Yaskawa INFORM job: OK_R2_O38-47,64(2)(90,0)_HARDOX.JBI

/JOB
//NAME OK_R2_O38-47,64(2)(90,0)_HARDOX
///FOLDERNAME X4
//POS
///NPOS 526,526,526,27,0,0
///TOOL 0
///POSTYPE PULSE
///PULSE
C00000=-102904,-190754,-108658,-56793,33718,43054
C00001=-112112,-124440,-79629,-37912,40591,30924
C00002=-145621,-43895,-45824,-14341,74181,8322
C00003=-153971,-33006,-36006,-12070,72386,5523
C00004=-155060,-28858,-31777,-11788,71762,5195
C00005=-155060,-28697,-30772,-11821,71236,5249
C00006=-155060,-28799,-31389,-11800,71558,5216
C00007=-155039,-34474,-35187,-11843,70998,5279
C00008=-155039,-34310,-34280,-11875,70534,5325
C00009=-155401,-30968,-32059,-11745,70828,5164
C00010=-155377,-31193,-32210,-11754,70809,5175
C00011=-155377,-31138,-31906,-11765,70652,5191
C00012=-155377,-31202,-32269,-11753,70839,5173
C00013=-155039,-34366,-34582,-11864,70687,5310
C00014=-155039,-34238,-33894,-11889,70337,5345
C00015=-155199,-32420,-32682,-11831,70497,5273
C00016=-155039,-34561,-35687,-11827,71256,5253
C00017=-155039,-34852,-37545,-11764,60729,-61899
C00018=-154233,-9766,-49045,-10778,79336,-63369
C00019=-160860,20388,-27147,4890,89580,-62573
C00020=-159005,21387,-26719,10091,95401,40718
C00021=-157683,11153,-31727,14818,95267,42221
C00022=-157333,10978,-31290,14718,94862,42282
C00023=-157333,10579,-30718,14700,94322,42218
C00024=-157333,10654,-30827,14702,94424,42231
C00025=-157208,13112,-28644,14670,94325,42258
C00026=-157333,10654,-30827,14702,94424,42231
C00027=-155197,18382,-25631,10360,99317,42541
C00028=-156128,18351,-25710,10541,99457,42258
C00029=-155197,18405,-25661,10361,99347,42543
C00030=-157150,29334,-18312,13637,104284,-74335
C00031=-160757,60877,11500,15991,103565,-75216
C00032=-161248,60365,12974,15966,102528,-75520
C00033=-161248,59958,13544,15927,101988,-75592
C00034=-161248,60034,13428,15935,102095,-75578
C00035=-161237,57406,10441,15969,102563,-75510
C00036=-161248,60034,13428,15935,102095,-75578
C00037=-165275,44513,292,24456,94477,-76762
C00038=-164215,44651,439,24212,94172,-76462
C00039=-165275,45390,-990,24520,95610,-76527
C00040=-163079,30136,-11541,1568,89602,-59565
C00041=-168249,10711,-29896,3021,91050,-61145
C00042=-157831,-12146,-38438,-15492,88791,-34391
C00043=-155039,-34561,-35687,-11827,71256,5253
C00044=-150032,-44426,-43245,-13273,71622,7027
C00045=-145621,-43895,-45824,-14341,74181,8322
C00046=-126188,-124725,-79701,-29915,35046,24780
C00047=-126055,-123557,-80227,-30584,36919,-46840
C00048=-134159,-82950,-60455,-26786,53755,-58167
C00049=-139895,-66772,-53027,-23260,55430,-61177
C00050=-141080,-64871,-50726,-22849,54691,-61528
C00051=-141080,-64256,-48906,-23069,53949,-61354
C00052=-141080,-64445,-49458,-23002,54172,-61405
C00053=-141699,-58855,-46559,-22430,55006,-61872
C00054=-141699,-58644,-45888,-22510,54724,-61808
C00055=-141384,-60956,-47106,-22771,54406,-61595
C00056=-141666,-61047,-48744,-22388,55219,-61905
C00057=-175822,-56342,-55375,-14128,52086,-76708
C00058=-175822,-56190,-54452,-14221,51611,-76640
C00059=-175822,-55829,-52499,-14419,50624,-76498
C00060=-175822,-55911,-52925,-14375,50838,-76529
C00061=-175468,-48992,-48997,-14371,52005,-76544
C00062=-175468,-48914,-48510,-14420,51752,-76509
C00063=-175508,-50972,-49701,-14458,51431,-76479
C00064=-175513,-50711,-51459,-14225,52610,-76651
C00065=-145967,-74518,-63848,-31232,56636,-64447
C00066=-145831,-74953,-63116,-31520,56106,-64204
C00067=-145831,-74483,-61568,-31767,55497,-64004
C00068=-145831,-74555,-61804,-31730,55589,-64033
C00069=-146027,-71690,-60453,-31425,56067,-64284
C00070=-145831,-74555,-61804,-31730,55589,-64033
C00071=-144274,-73926,-61511,-32332,56303,-63536
C00072=-142723,-73317,-61225,-32917,57019,-63047
C00073=-144274,-74241,-62562,-32164,56716,-63675
C00074=-154468,-41208,-54710,-20041,83622,-74370
C00075=-154754,-41232,-53805,-19994,83017,-74368
C00076=-154754,-41278,-52810,-20016,82420,-74271
C00077=-154754,-41268,-53081,-20010,82580,-74296
C00078=-154720,-44115,-54834,-20034,82227,-74224
C00079=-154754,-41268,-53081,-20010,82580,-74296
C00080=-155675,-41399,-53162,-19802,82346,-74583
C00081=-157197,-41522,-53239,-19453,81973,-75060
C00082=-155675,-41327,-54458,-19774,83133,-74712
C00083=-153395,-74759,-74503,-20498,79124,-73228
C00084=-153314,-74128,-71798,-20600,77886,-72984
C00085=-153314,-73934,-70558,-20645,77263,-72875
C00086=-153314,-73981,-70840,-20635,77403,-72900
C00087=-153337,-77229,-72353,-20684,76704,-72788
C00088=-153314,-73981,-70840,-20635,77403,-72900
C00089=-154242,-74168,-70928,-20438,77132,-73193
C00090=-156115,-74593,-71128,-20032,76581,-73782
C00091=-154242,-74289,-71704,-20409,77523,-73260
C00092=-153903,-106822,-81190,-17417,50996,-69253
C00093=-154273,-105923,-79990,-17297,50655,-69359
C00094=-154273,-105262,-78653,-17414,50193,-69275
C00095=-154273,-105373,-78877,-17395,50270,-69289
C00096=-154522,-102445,-77859,-17058,51058,-69542
C00097=-154273,-105373,-78877,-17395,50270,-69289
C00098=-152960,-105275,-78843,-18047,50584,-68754
C00099=-150354,-104788,-78676,-19283,51319,-67719
C00100=-152960,-106026,-80369,-17910,51111,-68853
C00101=-102904,-190754,-108658,-56793,33718,43054
C00102=-131529,-189509,-110128,-36771,24434,27261
C00103=-124211,-86804,-80218,-19393,77786,15538
C00104=-160160,17664,-548,-10057,75687,3034
C00105=-160660,22954,7322,-10002,73531,3037
C00106=-166196,35697,21074,-8411,71011,1264
C00107=-166196,35823,21925,-8432,70556,1296
C00108=-166196,35779,21629,-8424,70714,1284
C00109=-166257,29532,15350,-8374,71357,1216
C00110=-166257,29595,15824,-8387,71101,1234
C00111=-166146,32147,18367,-8436,70861,1292
C00112=-166154,31970,18190,-8433,70878,1288
C00113=-166154,32007,18455,-8439,70734,1299
C00114=-166154,31970,18190,-8433,70878,1288
C00115=-166179,28892,15129,-8411,71174,1259
C00116=-166179,28962,15640,-8424,70899,1278
C00117=-166104,30948,17607,-8456,70718,1318
C00118=-166176,28573,11657,-8324,73127,1123
C00119=-182178,81885,43168,-17852,83199,-7398
C00120=-187829,78862,41539,-16297,81531,-9102
C00121=-187829,78684,42370,-16320,80951,-9022
C00122=-187829,78533,43217,-16344,80374,-8946
C00123=-187829,78564,43028,-16338,80502,-8962
C00124=-188354,71817,34916,-16132,81866,-9324
C00125=-188354,71755,35176,-16139,81682,-9298
C00126=-188062,74943,38982,-16246,81057,-9118
C00127=-188087,74664,38647,-16237,81113,-9134
C00128=-188087,74606,38940,-16246,80911,-9107
C00129=-188087,74636,38787,-16240,81016,-9121
C00130=-188430,70936,34375,-16113,81733,-9334
C00131=-188430,70865,34684,-16121,81516,-9305
C00132=-188196,73082,37320,-16205,81097,-9170
C00133=-188430,71276,33065,-16084,82678,-9458
C00134=-165319,19573,3695,-8574,73487,1399
C00135=-163582,7043,-11027,-8999,76267,1804
C00136=-162101,-9402,-41897,-5301,86162,910
C00137=-133469,39121,-1061,931,85072,6891
C00138=-135751,46408,8355,1655,83056,6142
C00139=-135516,49476,14058,1587,81119,6193
C00140=-135516,49311,14679,1588,80652,6188
C00141=-135036,46950,11602,1434,81323,6352
C00142=-134946,46723,11962,1405,80982,6377
C00143=-135074,47950,13285,1445,80801,6333
C00144=-135102,44394,8734,1452,81774,6335
C00145=-133469,39121,-1061,931,85072,6891
C00146=-135146,16919,-22910,1456,87131,6386
C00147=-160578,-137207,-111137,27103,45167,-7155
C00148=-166532,-153428,-115250,33739,42272,-11545
C00149=-166532,-153428,-115250,33739,42272,-11545
C00150=-160883,-131526,-133102,-3483,78120,-6366
C00151=-103370,-159686,-136025,-1765,64172,-8056
C00152=-97179,-138237,-129333,-10238,76593,11306
C00153=-96065,-128281,-122439,-10507,77596,11607
C00154=-96065,-128106,-120653,-10546,76604,11690
C00155=-96065,-128281,-122439,-10507,77596,11607
C00156=-96974,-121186,-120234,-10189,79734,11117
C00157=-96065,-128281,-122439,-10507,77596,11607
C00158=-80019,-98046,-111669,-14399,88698,15911
C00159=-80077,-97852,-111516,-14385,88694,15892
C00160=-80077,-98331,-110658,-14385,87944,15982
C00161=-80077,-97897,-111441,-14385,88627,15900
C00162=-80867,-94680,-110202,-14197,89359,15553
C00163=-80077,-97897,-111441,-14385,88627,15900
C00164=-77060,-103837,-123440,-15157,93336,16325
C00165=-77104,-103620,-123385,-15148,93404,16303
C00166=-82212,-117279,-126602,-8714,87753,18646
C00167=-83304,-119533,-127995,-7425,87342,19011
C00168=-83304,-120285,-126924,-7427,86307,19072
C00169=-83304,-120125,-127175,-7427,86540,19060
C00170=-84285,-114583,-125380,-7184,88184,18645
C00171=-83304,-120125,-127175,-7427,86540,19060
C00172=-78124,-131037,-133000,-8681,85036,20864
C00173=-78124,-131037,-133000,-8681,85036,20864
C00174=-80781,-132367,-131851,-8063,83392,20088
C00175=-80781,-132658,-130737,-8071,82565,20142
C00176=-80781,-132579,-131090,-8068,82820,20125
C00177=-82215,-124520,-128659,-7695,85306,19491
C00178=-80136,-136061,-133167,-8229,82377,20371
C00179=-80218,-134686,-135534,-8183,84509,20204
C00180=-75563,-118157,-129697,-13391,92336,27261
C00181=-84024,-123631,-127734,-11595,87159,24981
C00182=-84024,-123979,-126960,-11598,86516,25042
C00183=-84024,-123746,-127494,-11596,86956,25000
C00184=-85048,-122093,-126977,-11373,87337,24623
C00185=-81994,-135324,-132084,-12059,84184,25946
C00186=-81994,-133752,-136174,-12028,87438,25630
C00187=-81994,-133752,-136174,-12028,87438,25630
C00188=-83107,-120864,-125937,-11789,87596,25245
C00189=-83880,-119254,-122492,-11630,86222,25116
C00190=-83880,-119583,-121326,-11637,85351,25197
C00191=-83880,-119399,-122020,-11633,85865,25149
C00192=-85062,-113328,-120022,-11369,87556,24598
C00193=-83880,-119399,-122020,-11633,85865,25149
C00194=-83464,-119333,-123502,-11716,86850,25194
C00195=-84085,-116294,-122008,-11580,87393,24935
C00196=-84085,-116863,-120480,-11583,86184,25047
C00197=-84085,-116689,-121008,-11580,86590,25010
C00198=-85140,-111307,-119205,-11348,88071,24523
C00199=-84085,-116194,-122230,-11576,87577,24918
C00200=-82864,-118268,-130611,-11862,91757,24924
C00201=-82864,-118268,-130611,-11862,91757,24924
C00202=-86851,-110557,-120071,-10968,88745,23893
C00203=-86851,-111341,-118540,-10968,87421,24011
C00204=-86851,-110811,-119621,-10968,88345,23929
C00205=-88598,-109546,-119189,-10575,88500,23337
C00206=-86851,-110811,-119621,-10968,88345,23929
C00207=-83825,-124590,-131318,-11630,88867,24881
C00208=-82909,-127853,-136097,-11834,90233,25054
C00209=-84148,-125178,-125504,-11579,85018,25131
C00210=-81186,-118241,-121828,-12198,86718,25964
C00211=-81186,-118533,-120824,-12201,85966,26037
C00212=-81186,-118483,-121017,-12200,86107,26023
C00213=-82314,-113243,-119285,-11952,87535,25506
C00214=-81186,-118241,-121828,-12198,86718,25964
C00215=-87931,-140644,-131144,-10841,80108,24284
C00216=-89960,-139833,-128047,-10433,78377,23732
C00217=-89960,-139550,-127065,-10448,77925,23770
C00218=-89960,-139622,-127307,-10444,78035,23761
C00219=-90753,-134395,-125809,-10209,79670,23349
C00220=-89456,-143397,-129529,-10578,77538,23979
C00221=-95203,-107502,-133483,-6717,98684,21003
C00222=-95203,-107502,-133483,-6717,98684,21003
C00223=70091,-137861,-134613,19540,89589,-11549
C00224=70091,-137861,-134613,19540,89589,-11549
C00225=89914,-142582,-130695,14485,81723,-10120
C00226=90202,-137048,-128128,14398,82897,-9883
C00227=90202,-136718,-126391,14423,82025,-9985
C00228=90202,-136862,-127082,14413,82365,-9945
C00229=91010,-131454,-125503,14223,83978,-9478
C00230=90202,-137070,-128271,14397,82970,-9874
C00231=76195,-137070,-128271,14397,82970,-9874
C00232=74994,-123934,-123423,14560,86840,-9835
C00233=74994,-124092,-122198,14564,86029,-9931
C00234=74994,-124005,-122955,14561,86525,-9872
C00235=76141,-119465,-121513,14342,87728,-9340
C00236=72631,-133219,-128550,14998,85696,-10781
C00237=72631,-131663,-134232,14989,89852,-10278
C00238=50716,-132590,-134806,14983,95067,-21778
C00239=53786,-122460,-125023,14607,93736,-20890
C00240=54881,-121663,-124068,14472,93371,-20558
C00241=54881,-122014,-122728,14450,92397,-20672
C00242=54881,-121856,-123398,14460,92875,-20616
C00243=56721,-117465,-121986,14267,93906,-19868
C00244=54881,-121856,-123398,14460,92875,-20616
C00245=55322,-120745,-123309,14420,93300,-20415
C00246=55322,-120747,-123302,14420,93295,-20416
C00247=55322,-120978,-122461,14407,92679,-20487
C00248=55322,-120864,-122902,14414,92999,-20450
C00249=56710,-117554,-121835,14266,93775,-19889
C00250=54436,-122887,-123768,14509,92662,-20793
C00251=54436,-122067,-126198,14556,94519,-20574
C00252=53688,-126302,-127242,14482,93230,-21000
C00253=7968,-117738,-135568,14910,102458,-19890
C00254=7968,-117738,-135568,14910,102458,-19890
C00255=4119,-116606,-125698,15061,97809,-21757
C00256=7770,-114903,-122318,14590,96007,-20739
C00257=7770,-115418,-121244,14557,95111,-20843
C00258=7770,-115024,-122084,14598,95810,-20761
C00259=9375,-110655,-120613,14452,96836,-20097
C00260=7770,-115024,-122084,14598,95810,-20761
C00261=10569,-102485,-118509,17167,107955,-30726
C00262=17008,-101176,-116544,17116,107524,-30934
C00263=-121481,-92648,-105286,-5369,115019,-86755
C00264=-120615,-96829,-107734,-5213,114434,-86412
C00265=23859,-150611,-131722,11614,81196,-13147
C00266=5605,-98558,-114313,9016,91646,-19053
C00267=5292,-97369,-113802,9089,91971,-19129
C00268=5881,-109040,-123705,8960,92007,-18939
C00269=6434,-120006,-133010,8839,92040,-18760
C00270=-12667,-120051,-129788,-19636,91452,63850
C00271=-15640,-171133,-136982,-20070,70138,66271
C00272=3779,-163113,-125940,-36463,74354,73480
C00273=-120436,-95190,-80290,-14692,43277,16053
C00274=-119715,-95468,-78930,-15521,42464,16563
C00275=1349,-140937,-118482,-38247,78517,71026
C00276=-15636,-141614,-117585,-35447,65083,67762
C00277=-17609,-126505,-112505,-34601,67163,66072
C00278=-24043,-118481,-124771,-21586,79008,61529
C00279=-24043,-118481,-124771,-21586,79008,61529
C00280=-75030,-118005,-124618,-21594,79160,61521
C00281=-115715,-153549,-128562,15788,54400,49074
C00282=-122131,-153692,-122292,24372,49463,44977
C00283=-120438,-96789,-101713,-1489,48968,3516
C00284=-120356,-99154,-104149,-1548,49253,3547
C00285=-84198,-116806,-111213,1772,54897,61304
C00286=-87160,-120534,-109364,10018,48087,58269
C00287=-90828,-138253,-118809,13315,45388,56216
C00288=-90828,-138253,-118809,13315,45388,56216
C00289=-90828,-142934,-129815,12421,49655,56806
C00290=-90829,-142933,-129813,12421,49658,56806
C00291=-119872,-163920,-132846,33283,49576,42941
C00292=-126991,-146326,-124104,35016,55490,41598
C00293=-120835,-94912,-106201,4597,84031,3620
C00294=-120296,-100536,-106811,4468,81494,3706
C00295=-119922,-143587,-123205,31413,53438,44308
C00296=-77415,-98459,-105381,5383,51560,63214
C00297=-71925,-92447,-101662,533,50488,65336
C00298=-77718,-122737,-116129,5642,44048,62545
C00299=-53268,-154266,-130714,-22807,48565,72872
C00300=-53268,-154266,-130714,-22807,48565,72872
C00301=-65704,-162398,-123942,-17029,37659,69009
C00302=-69631,-160797,-117543,-19584,31037,68677
C00303=-120621,-91661,-79831,4809,93096,-80691
C00304=-120610,-95504,-82099,4805,92519,-80709
C00305=-64928,-151300,-115352,-22074,35531,70301
C00306=-55359,-110208,-106429,-19631,55099,70468
C00307=-56474,-111761,-106561,-17625,52293,70865
C00308=-58794,-112885,-105581,-13565,47681,71177
C00309=-50265,-141050,-116073,-27906,38980,77613
C00310=-41790,-175398,-134696,-41509,59591,72504
C00311=-40096,-167295,-132799,-40833,62675,71982
C00312=-66805,-175580,-133819,-17842,44997,58057
C00313=-120613,-98309,-97516,-18774,58387,20033
C00314=-120296,-100165,-96633,-19249,57041,20409
C00315=-66730,-175408,-133780,-17867,45074,58078
C00316=-65136,-170814,-132569,-18309,46965,58464
C00317=-52364,-139651,-124628,-28315,65404,66743
C00318=-50532,-107164,-114440,-27328,75285,64992
C00319=-50521,-107002,-114383,-27326,75331,64985
C00320=-56147,-114427,-116211,-21096,65709,65656
C00321=-54523,-105936,-113271,-21470,68505,65739
C00322=-49750,-132075,-132074,-23871,68057,67633
C00323=-51888,-141517,-135531,-28423,71943,65142
C00324=-58410,-142164,-121837,-32385,67064,69630
C00325=-58892,-132878,-117266,-33819,71370,71170
C00326=-120621,-92022,-79948,-5717,93324,-87803
C00327=-120611,-95871,-82213,-5711,92744,-87773
C00328=-91898,-177824,-128316,2778,37745,41927
C00329=-76561,-127099,-115440,3526,55962,41360
C00330=-98908,-102884,-107387,29228,75304,22104
C00331=-100715,-115554,-120696,29641,77391,21955
C00332=-99511,-125054,-130815,29118,78165,22610
C00333=30978,-142903,-136378,16839,87530,-25088
C00334=48053,-137432,-126920,10736,83825,-19877
C00335=-120514,-92773,-72492,63824,26217,-40707
C00336=-122096,-91517,-72885,63277,27653,-40461
C00337=46723,-132150,-125263,10235,84639,-20316
C00338=38144,-96146,-111322,6693,87070,-23612
C00339=36690,-89699,-108774,7082,88920,-23976
C00340=38688,-150385,-135608,6755,74185,-24124
C00341=34744,-121097,-133452,9828,92546,-23976
C00342=92930,-150385,-135608,6755,74185,-24124
C00343=107101,-138400,-125652,2740,73384,-19202
C00344=-120610,-93305,-77258,53115,31058,22991
C00345=-120294,-94166,-75974,54567,30127,22239
C00346=116035,-135916,-124846,-7405,75208,-6894
C00347=75429,-100276,-113037,4073,85400,-20589
C00348=88876,-89136,-108695,-11365,90939,-2676
C00349=92139,-118134,-128268,-12138,88585,-1394
C00350=96790,-150711,-134355,-17072,70659,2161
C00351=96790,-150711,-134355,-17072,70659,2161
C00352=652,-114254,-134536,-4800,91191,-3391
C00353=-166532,-153428,-115250,33739,42272,-11545
C00354=-166532,-153428,-115250,33739,42272,-11545
C00355=-124114,-84683,-61597,-48557,28871,-52530
C00356=-120672,9825,17632,-53753,29009,-53309
C00357=-120673,9828,17635,-53752,29009,-53309
C00358=-119969,9889,17391,-53999,29527,-53154
C00359=-120673,10502,19535,-54974,28515,-52685
C00360=-120213,7916,15945,-54003,29309,-53162
C00361=-120673,9268,16917,-53528,29103,-53422
C00362=-120673,9346,17029,-53570,29085,-53403
C00363=-120325,9631,17167,-53735,29324,-53303
C00364=-120673,9869,17671,-53754,29008,-53308
C00365=-120672,9864,17667,-53755,29008,-53308
C00366=-124114,-84683,-61597,-48557,28871,-52530
C00367=-131339,-154294,-79414,-109628,16862,-24377
C00368=-234701,-24447,-54419,57638,71697,57534
C00369=-192045,-4471,-49137,31395,56880,70337
C00370=-172212,48807,-7818,-1281,85806,67502
C00371=-182022,60397,16725,362,120111,76099
C00372=-181268,75249,48221,-1582,120068,76073
C00373=-181298,74023,48403,-1581,119325,76072
C00374=-181356,72617,44998,-1625,120698,76029
C00375=-181183,75410,49585,-1539,119314,76118
C00376=-180620,73123,47328,-1344,119537,76335
C00377=-180498,74390,47192,-1310,120274,76376
C00378=-180299,81057,52347,-1242,120531,76452
C00379=-174789,63735,852,-597,96026,66536
C00380=-179792,32070,-16354,13350,79915,65662
C00381=-186878,-39073,-38836,41246,34970,63358
C00382=-188022,-31651,-32655,42206,35520,62864
C00383=-188256,-32514,-32154,43117,35074,62369
C00384=-188651,-34827,-34931,42941,35654,62475
C00385=-186847,-32376,-33139,41284,34905,63337
C00386=-187464,-35744,-36703,41375,35550,63305
C00387=-188726,-40923,-42933,41373,37038,63352
C00388=-176527,13729,-19852,11997,65990,74911
C00389=-182239,28447,-8651,22613,76038,76180
C00390=-177930,36952,-84,19488,73368,78350
C00391=-155197,18405,-25661,10361,99347,42543
C00392=-157150,29334,-18312,13637,104284,-74335
C00393=-160757,60877,11500,15991,103565,-75216
C00394=-163498,59946,10428,16358,104233,-76035
C00395=-164943,57615,11020,16171,102868,-76491
C00396=-161151,58385,12228,17218,102481,-74998
C00397=-161151,58385,12228,17218,102481,-74998
C00398=-165789,43027,488,27315,92842,-76690
C00399=-160186,27839,-15652,14617,84558,-74255
C00400=-160167,20989,-21384,10653,80805,-75466
C00401=-147415,42895,344,-1586,77779,-65108
C00402=-147415,42895,344,-1586,77779,-65108
C00403=-160856,55961,7713,8964,101583,-87584
C00404=-164943,57615,11020,16171,102868,-76491
C00405=-164893,58388,10563,16217,103512,-76386
C00406=-167418,31456,-19601,16982,108508,-76513
C00407=-168563,-3240,-51288,17325,110317,-76617
C00408=-137180,-42892,-79374,12190,102290,-67498
C00409=-196569,5763,-30645,36969,53415,67065
C00410=-234701,-24447,-54419,57638,71697,57534
C00411=-149956,-143190,-113193,-9671,18752,-75469
C00412=-134160,-28568,-62536,-18892,48395,-71822
C00413=-120672,9794,17604,-61241,37188,-52240
C00414=-120672,9794,17604,-61241,37188,-52240
C00415=-120555,9400,17043,-61125,37334,-52300
C00416=-120673,9158,15746,-60306,37604,-52768
C00417=-120213,7880,15913,-61361,37506,-52152
C00418=-120673,9106,16782,-61064,37264,-52340
C00419=-120673,9123,16797,-61065,37265,-52339
C00420=-120025,10235,17860,-61424,37632,-52107
C00421=-120673,9754,17568,-61239,37189,-52241
C00422=-120672,9754,17569,-61239,37189,-52241
C00423=-134138,-28506,-62498,-18910,48408,-71815
C00424=-154186,-159927,-117173,-847,12331,-79725
C00425=-85861,-99082,-105113,-44329,59147,-50836
C00426=-83984,-106882,-107996,-46165,58479,-49488
C00427=-120674,-14372,-36148,-15341,86455,-69375
C00428=-120676,-10921,-33498,-15340,86592,-69392
C00429=-120687,11625,-15842,-15708,100514,-71147
C00430=-121175,-12454,-34682,-15229,86445,-69544
C00431=-120675,-14159,-37235,-15335,87207,-69469
C00432=-123028,8470,-18643,-15581,100180,-71911
C00433=-120676,-11639,-34054,-15340,86566,-69391
C00434=-120674,-14390,-36162,-15341,86455,-69375
C00435=-120676,-14354,-36134,-15765,85734,14225
C00436=-120676,-14354,-36134,-15765,85734,14225
C00437=-120800,8775,-20209,-16101,100075,12323
C00438=-120676,-14158,-37234,-15757,86484,14129
C00439=-120165,-16255,-37568,-15883,85739,14397
C00440=-123278,5465,-23101,-15908,99682,11524
C00441=-120676,-14374,-36149,-15765,85733,14224
C00442=-120676,-14373,-36148,-15765,85733,14225
C00443=-98406,-95981,-107671,-30899,65126,-72820
C00444=-145831,-74953,-63116,-31520,56106,-64204
C00445=-144848,-71159,-60112,-31747,56614,-63934
C00446=-154467,-73379,-61267,-27433,52858,-67287
C00447=-154467,-73379,-61267,-27433,52858,-67287
C00448=-156206,-49547,-56219,-21205,75840,-73631
C00449=-164648,-31551,-50013,-8827,90724,-77034
C00450=-170479,-23568,-45543,1063,96292,-78073
C00451=-166074,-24155,-45964,927,96422,-76584
C00452=-166074,-24155,-45964,927,96422,-76584
C00453=-175560,-40435,-53688,14531,84002,-78896
C00454=-144848,-71159,-60112,-31747,56614,-63934
C00455=-145051,-72959,-63458,-31286,57513,-64321
C00456=-138712,-107565,-77308,-37350,52342,-59302
C00457=-138851,-102977,-73181,-37386,52136,-59285
C00458=-151617,-106240,-74249,-32666,46092,-63553
C00459=-151617,-106240,-74249,-32666,46092,-63553
C00460=-162721,-86144,-76024,-13696,67242,-72648
C00461=-162970,-63526,-68628,-11422,86228,-74954
C00462=-173294,-52958,-64274,1686,93665,-76737
C00463=-167662,-54364,-65065,1153,93332,-74867
C00464=-167662,-54364,-65065,1153,93332,-74867
C00465=-172379,-78924,-74785,7773,74246,-76598
C00466=-138851,-102977,-73181,-37386,52136,-59285
C00467=-139567,-106681,-78131,-36615,52754,-59917
C00468=-98406,-95981,-107671,-30899,65126,25478
C00469=-97498,-103141,-110365,-31836,63713,26282
C00470=-158741,-152165,-85078,-53213,16407,-64133
C00471=-151185,-64492,-56891,-27025,41971,-76525
C00472=-187574,37417,13419,2960,77279,72462
C00473=-187020,38831,14880,2796,77088,72647
C00474=-180715,58337,34412,-9745,85564,73616
C00475=-187315,39588,15664,2886,77004,72543
C00476=-187570,37474,12233,2951,78037,72481
C00477=-180152,63979,41102,-12031,86543,73575
C00478=-187574,37421,13424,2960,77279,72462
C00479=-187576,37412,13414,2961,77280,72461
C00480=-187610,37331,13331,3255,76507,-7692
C00481=-182719,57686,35499,-3659,79600,-3173
C00482=-182518,60502,39600,-3732,78534,-3072
C00483=-187825,35310,11263,3318,76749,-7758
C00484=-187564,37491,12251,3232,77251,-7657
C00485=-186882,65081,44973,-2747,77404,-4541
C00486=-187574,37420,13423,3244,76495,-7680
C00487=-174916,2091,-20307,-7000,70210,-31977
C00488=-151185,-64492,-56891,-27025,41971,-76525
C00489=-158741,-152165,-85078,-53213,16407,-64133
C00490=-136335,-97157,-88666,-6240,65884,-69249
C00491=-141826,-62430,-72987,-3929,73707,-71532
C00492=-140052,-21130,-52867,24635,78479,-75610
C00493=-137473,58120,11150,19511,106253,-71077
C00494=-132799,89049,47439,16428,114143,-68872
C00495=-132090,97611,56676,15970,118552,-68089
C00496=-132278,96746,56340,15749,120045,-68002
C00497=-135984,107314,69748,14048,119719,-69614
C00498=-135785,103774,66356,14147,119946,-69504
C00499=-131685,106105,70627,22443,116548,-67586
C00500=-133954,98465,50155,16232,124944,-67916
C00501=-142400,32764,-15276,22713,92529,-74169
C00502=-109290,70352,15308,-18647,88059,-61302
C00503=-83699,85527,52785,-52979,68456,-51263
C00504=-80420,18251,15496,-64356,57036,-45994
C00505=-80421,18253,15498,-64356,57035,-45994
C00506=-80345,19089,16149,-64356,57099,-45998
C00507=-80421,18695,17178,-64825,56670,-45601
C00508=-79680,17143,14466,-64475,57547,-45892
C00509=-77910,31513,28141,-65399,58243,-45083
C00510=-78671,21218,15982,-64051,58734,-46270
C00511=-89230,-40025,-45988,-57168,55507,-51535
C00512=-165830,-102325,-81854,21592,21746,-90581
C00513=-143448,-1036,-52885,-16428,93385,-83560
C00514=-164922,35704,-16289,-11037,108697,-82216
C00515=-167627,32529,-19588,-10739,108771,-83097
C00516=-167991,31957,-18569,-11486,108743,-83384
C00517=-80421,18695,17178,-64825,56670,-45601
C00518=-79680,17143,14466,-64475,57547,-45892
C00519=-167646,32101,-18426,-11522,108769,-83275
C00520=-171644,46039,-4653,1010,116229,-75636
C00521=-161692,44011,-6873,1232,116433,-72213
C00522=-163610,51425,3446,12841,118918,-64739
C00523=-163510,54015,1682,13204,121259,-64411
C00524=-159201,-7258,-55066,4115,89555,-67128
C00525=-140583,-29745,-76270,-2898,90924,-61741
BC00000=155275,760074,251743
BC00001=155275,819591,251743
BC00002=155275,819591,251743
BC00003=155275,819591,251743
BC00004=155275,819591,251743
BC00005=155275,819591,251743
BC00006=155275,819591,251743
BC00007=155275,819591,251742
BC00008=155275,819591,251742
BC00009=155275,819591,251742
BC00010=155275,819591,251742
BC00011=155275,819591,251742
BC00012=155275,819591,251742
BC00013=155275,819591,251742
BC00014=155275,819591,251742
BC00015=155275,819591,251742
BC00016=155275,819591,251742
BC00017=155275,819591,251742
BC00018=141983,819591,71290
BC00019=141983,819591,71290
BC00020=141983,819591,71290
BC00021=141983,819591,71290
BC00022=141984,819591,71287
BC00023=141984,819591,71287
BC00024=141984,819591,71287
BC00025=141984,819591,71287
BC00026=141984,819591,71287
BC00027=141984,819591,71285
BC00028=141984,819591,71285
BC00029=141984,819591,71285
BC00030=141984,819591,71285
BC00031=165972,803410,43335
BC00032=165972,803410,43335
BC00033=165972,803410,43335
BC00034=165972,803410,43335
BC00035=165972,803410,43335
BC00036=165972,803410,43335
BC00037=165972,803410,43335
BC00038=165972,803410,43335
BC00039=165972,803410,43335
BC00040=163388,807319,93684
BC00041=163388,807319,93684
BC00042=160216,812118,155484
BC00043=155275,819591,251742
BC00044=155275,819591,251743
BC00045=155275,819591,251743
BC00046=155275,819591,251743
BC00047=155275,819591,251743
BC00048=155275,819591,251743
BC00049=155275,819591,251742
BC00050=155275,819591,251742
BC00051=155275,819591,251742
BC00052=155275,819591,251742
BC00053=155275,819591,251742
BC00054=155275,819591,251742
BC00055=155275,819591,251742
BC00056=155275,819591,251742
BC00057=189858,819605,176881
BC00058=189858,819605,176881
BC00059=189858,819605,176881
BC00060=189858,819605,176881
BC00061=189858,819605,176881
BC00062=189858,819605,176881
BC00063=189858,819605,176881
BC00064=189858,819605,176881
BC00065=189858,819605,176881
BC00066=189858,819605,176878
BC00067=189858,819605,176878
BC00068=189858,819605,176878
BC00069=189858,819605,176878
BC00070=189858,819605,176878
BC00071=189858,819605,176878
BC00072=189858,819605,176878
BC00073=189858,819605,176878
BC00074=189858,819605,176878
BC00075=189858,819605,176878
BC00076=189858,819605,176878
BC00077=189858,819605,176878
BC00078=189858,819605,176878
BC00079=189858,819605,176878
BC00080=189858,819605,176878
BC00081=189858,819605,176878
BC00082=189858,819605,176878
BC00083=189858,819605,176877
BC00084=189858,819605,176877
BC00085=189858,819605,176877
BC00086=189858,819605,176877
BC00087=189858,819605,176877
BC00088=189858,819605,176877
BC00089=189858,819605,176877
BC00090=189858,819605,176877
BC00091=189858,819605,176877
BC00092=189858,819605,176876
BC00093=189858,819605,176876
BC00094=189858,819605,176876
BC00095=189858,819605,176876
BC00096=189858,819605,176876
BC00097=189858,819605,176876
BC00098=189858,819605,176876
BC00099=189858,819605,176876
BC00100=189858,819605,176876
BC00101=155275,760074,251743
BC00102=334637,762746,239047
BC00103=334637,842186,239047
BC00104=334637,842186,239047
BC00105=334637,842186,239047
BC00106=334637,842186,239047
BC00107=334637,842186,239047
BC00108=334637,842186,239047
BC00109=334637,842186,239047
BC00110=334637,842186,239047
BC00111=334637,842186,239047
BC00112=334637,842186,239047
BC00113=334637,842186,239047
BC00114=334637,842186,239047
BC00115=334637,842186,239047
BC00116=334637,842186,239047
BC00117=334637,842186,239047
BC00118=334637,842186,239047
BC00119=355885,842186,63101
BC00120=355885,842187,63099
BC00121=355885,842187,63099
BC00122=355885,842187,63099
BC00123=355885,842187,63099
BC00124=355885,842187,63099
BC00125=355885,842187,63099
BC00126=355885,842187,63099
BC00127=355885,842187,63099
BC00128=355885,842187,63099
BC00129=355885,842187,63099
BC00130=355885,842187,63099
BC00131=355885,842187,63099
BC00132=355885,842187,63099
BC00133=355885,842187,63099
BC00134=334637,842186,239047
BC00135=334637,842186,239047
BC00136=336476,842187,209320
BC00137=343292,842193,99157
BC00138=343292,842193,99157
BC00139=343292,842193,99157
BC00140=343292,842193,99157
BC00141=343292,842193,99157
BC00142=343292,842193,99157
BC00143=343292,842193,99157
BC00144=343292,842193,99157
BC00145=343292,842193,99157
BC00146=343292,842193,99157
BC00147=343292,842193,99157
BC00148=343292,714597,99157
BC00149=343292,714597,1074810
BC00150=343292,714597,1074810
BC00151=343292,942381,1074810
BC00152=336034,956109,1074810
BC00153=336034,956109,1074810
BC00154=336034,956109,1074810
BC00155=336034,956109,1074810
BC00156=336034,956109,1074810
BC00157=336034,956109,1074810
BC00158=336034,956109,1074810
BC00159=336034,956109,1074810
BC00160=336034,956109,1074810
BC00161=336034,956109,1074810
BC00162=336034,956109,1074810
BC00163=336034,956109,1074810
BC00164=336034,956109,1074810
BC00165=371500,1003655,1072368
BC00166=371500,1011303,1072368
BC00167=371500,1012871,1072368
BC00168=371500,1012871,1072368
BC00169=371500,1012871,1072368
BC00170=371500,1012871,1072368
BC00171=371500,1012871,1072368
BC00172=371500,1012871,1072368
BC00173=310141,1007143,1071829
BC00174=310141,1007143,1071829
BC00175=310141,1007143,1071829
BC00176=310141,1007143,1071829
BC00177=310141,1007143,1071829
BC00178=310141,1007143,1071829
BC00179=310141,1007143,1071829
BC00180=246928,976807,1071829
BC00181=246928,976807,1071829
BC00182=246928,976807,1071829
BC00183=246928,976807,1071829
BC00184=246928,976807,1071829
BC00185=246928,976807,1071829
BC00186=246928,976807,1071829
BC00187=144012,964080,1063254
BC00188=144012,964080,1063254
BC00189=144012,964080,1063254
BC00190=144012,964080,1063254
BC00191=144012,964080,1063254
BC00192=144012,964080,1063254
BC00193=144012,964080,1063254
BC00194=107418,957008,1063254
BC00195=107418,957008,1063254
BC00196=107418,957008,1063254
BC00197=107418,957008,1063254
BC00198=107418,957008,1063254
BC00199=107418,957008,1063254
BC00200=107418,957008,1063254
BC00201=126016,899142,1063254
BC00202=126016,899142,1063254
BC00203=126016,899142,1063254
BC00204=126016,899142,1063254
BC00205=126016,899142,1063254
BC00206=126016,899142,1063254
BC00207=126016,899142,1063254
BC00208=32383,899142,1063254
BC00209=33723,949074,1063254
BC00210=33723,949074,1063254
BC00211=33723,949074,1063254
BC00212=33723,949074,1063254
BC00213=33723,949074,1063254
BC00214=33723,949074,1063254
BC00215=7047,944370,1063254
BC00216=6971,946386,1064283
BC00217=6971,946386,1064283
BC00218=6971,946386,1064283
BC00219=6971,946386,1064283
BC00220=6971,946386,1064283
BC00221=6971,946386,1064283
BC00222=25103,830564,1064283
BC00223=1840,976824,1064283
BC00224=1840,1022624,1064283
BC00225=1840,1022624,1064283
BC00226=1840,1022624,1064283
BC00227=1840,1022624,1064283
BC00228=1840,1022624,1064283
BC00229=1840,1022624,1064283
BC00230=1840,1022624,1064283
BC00231=32240,1021120,1065802
BC00232=32240,1021120,1065802
BC00233=32240,1021120,1065802
BC00234=32240,1021120,1065802
BC00235=32240,1021120,1065802
BC00236=32240,1021120,1065802
BC00237=32240,1021120,1065802
BC00238=75978,1001728,1065802
BC00239=75977,1001729,1065799
BC00240=75977,1001729,1065799
BC00241=75977,1001729,1065799
BC00242=75977,1001729,1065799
BC00243=75977,1001729,1065799
BC00244=75977,1001729,1065799
BC00245=117549,1001729,1065799
BC00246=117549,1001729,1065799
BC00247=117549,1001729,1065799
BC00248=117549,1001729,1065799
BC00249=117549,1001729,1065799
BC00250=117549,1001729,1065799
BC00251=117549,1001729,1065799
BC00252=56674,1036312,1065895
BC00253=56674,1036312,1065895
BC00254=30889,1102979,1065895
BC00255=45214,1102979,1065895
BC00256=45214,1102979,1065895
BC00257=45214,1102979,1065895
BC00258=45214,1102978,1065892
BC00259=45214,1102978,1065892
BC00260=45214,1102978,1065892
BC00261=45214,1102978,1065889
BC00262=45214,1102978,1065889
BC00263=145257,917701,1075175
BC00264=145257,917701,1075175
BC00265=45214,1102978,1065887
BC00266=45214,1102978,1065887
BC00267=45214,1102978,1065887
BC00268=45214,1102978,1065887
BC00269=45214,1102978,1065887
BC00270=50349,952936,1065887
BC00271=50349,952936,1065887
BC00272=50349,952936,1065887
BC00273=156935,778985,1075175
BC00274=156935,778985,1075175
BC00275=50349,952936,1065887
BC00276=72136,952936,1065887
BC00277=72136,952936,1065887
BC00278=72136,952936,1065887
BC00279=58646,939592,1065887
BC00280=33,880302,1065887
BC00281=33,928742,1065885
BC00282=33,928742,1065885
BC00283=369319,873480,1075175
BC00284=369319,873480,1075175
BC00285=33,928742,1065885
BC00286=33,928742,1065885
BC00287=33,928742,1065885
BC00288=33,926822,1072255
BC00289=33,849370,1070063
BC00290=271563,976879,1070062
BC00291=312671,982863,1065015
BC00292=312671,982863,1065015
BC00293=4086,859403,1075175
BC00294=4086,859403,1075175
BC00295=312671,982863,1065015
BC00296=312671,982863,1065015
BC00297=312671,982863,1065015
BC00298=312671,982863,1065015
BC00299=312671,982863,1065015
BC00300=280596,959851,1065015
BC00301=280596,959851,1065015
BC00302=280596,959851,1065015
BC00303=125992,771300,1075175
BC00304=125992,771300,1075175
BC00305=280596,959851,1065015
BC00306=280596,959851,1065012
BC00307=280596,959851,1065013
BC00308=280596,959851,1065015
BC00309=280596,959851,1065015
BC00310=280596,959851,1065015
BC00311=211687,973675,1065015
BC00312=204246,973675,1065015
BC00313=168833,851602,1075175
BC00314=168833,851602,1075175
BC00315=204246,973675,1065015
BC00316=204246,973675,1065015
BC00317=204246,973675,1065015
BC00318=204246,973675,1065015
BC00319=204246,973675,1065015
BC00320=204246,973675,1065015
BC00321=204246,973675,1065015
BC00322=204246,973675,1065015
BC00323=93803,958451,1065015
BC00324=93803,958451,1065015
BC00325=93804,958451,1065014
BC00326=27668,771045,1075175
BC00327=27668,771045,1075175
BC00328=93804,958451,1065014
BC00329=93804,958451,1065014
BC00330=93804,958451,1065014
BC00331=93804,958451,1065014
BC00332=93804,958451,1065014
BC00333=58899,987526,1068118
BC00334=58899,987526,1068118
BC00335=345503,839022,1075175
BC00336=345503,839022,1075175
BC00337=58899,987526,1068118
BC00338=58899,987526,1068118
BC00339=58899,987526,1068118
BC00340=58899,987526,1068118
BC00341=58139,987526,1068216
BC00342=1984,1028862,1068118
BC00343=1984,1028862,1068118
BC00344=310150,835828,1075175
BC00345=310150,835828,1075175
BC00346=1984,1028862,1068118
BC00347=1984,1028862,1068118
BC00348=1984,1028862,1068118
BC00349=1984,1028862,1068118
BC00350=1984,1028862,1068118
BC00351=1984,833796,1068118
BC00352=56336,759226,1064779
BC00353=343292,714597,1074810
BC00354=343292,714597,99157
BC00355=326718,829986,221879
BC00356=326019,834851,227054
BC00357=323796,839870,208138
BC00358=322906,841877,200572
BC00359=322906,841877,200572
BC00360=322906,841877,200572
BC00361=327037,844194,200572
BC00362=331719,846821,200572
BC00363=335850,849138,200572
BC00364=336739,847130,208139
BC00365=338963,842112,227055
BC00366=326718,829986,221879
BC00367=326718,721817,221879
BC00368=301908,735078,53
BC00369=301908,735078,53
BC00370=257340,761494,53
BC00371=218510,827652,130053
BC00372=218510,827652,130053
BC00373=218510,827652,130053
BC00374=218510,827652,130053
BC00375=218510,827652,130053
BC00376=218510,827652,130053
BC00377=218510,827652,130053
BC00378=218510,827652,130053
BC00379=257340,761494,53
BC00380=243122,776164,27952
BC00381=213981,806232,85133
BC00382=213981,806232,85133
BC00383=213981,806232,85133
BC00384=213981,806232,85133
BC00385=213981,806232,85133
BC00386=213981,806232,85133
BC00387=213981,806232,85133
BC00388=213981,806232,85133
BC00389=213981,806232,85133
BC00390=213981,806232,85133
BC00391=141984,819591,71285
BC00392=141984,819591,71285
BC00393=165972,803410,43335
BC00394=165972,803410,43335
BC00395=166113,803418,43458
BC00396=166113,803418,43458
BC00397=166113,803418,43458
BC00398=166113,803418,43458
BC00399=166113,803418,43458
BC00400=166113,803418,43458
BC00401=145810,765805,43458
BC00402=145810,765805,43458
BC00403=166112,803416,43457
BC00404=166113,803418,43458
BC00405=166113,803418,43458
BC00406=166113,803418,43458
BC00407=166113,803418,43458
BC00408=166113,803418,43458
BC00409=301908,735078,53
BC00410=301908,735078,53
BC00411=326019,716112,4997
BC00412=326019,754467,4997
BC00413=315535,829024,226895
BC00414=312111,833369,207979
BC00415=310742,835107,200413
BC00416=310742,835107,200413
BC00417=310742,835107,200413
BC00418=306612,832790,200413
BC00419=301791,830087,200413
BC00420=297661,827770,200413
BC00421=299030,826032,207979
BC00422=302454,821686,226895
BC00423=326019,802314,4997
BC00424=326019,740906,5323
BC00425=131939,688818,32608
BC00426=131939,774315,32608
BC00427=131939,801396,210359
BC00428=131334,801067,183577
BC00429=131093,800936,172865
BC00430=131093,800936,172865
BC00431=131093,800936,172865
BC00432=131093,800936,172865
BC00433=125276,797669,183577
BC00434=125880,797998,210358
BC00435=132304,800008,176562
BC00436=128880,804353,157646
BC00437=127511,806091,150080
BC00438=127511,806091,150080
BC00439=127511,806091,150080
BC00440=127511,806091,150080
BC00441=122408,800723,157646
BC00442=125832,796378,176562
BC00443=132304,777362,53
BC00444=189858,819605,176878
BC00445=189788,819557,176486
BC00446=189756,819535,176304
BC00447=189756,819535,176304
BC00448=189756,819535,176304
BC00449=189756,819535,176304
BC00450=189690,819490,175931
BC00451=189690,819490,175931
BC00452=189690,819490,175931
BC00453=189690,819490,175931
BC00454=189788,819557,176486
BC00455=189788,819557,176486
BC00456=189788,819557,176486
BC00457=189788,819557,176486
BC00458=189788,819557,176485
BC00459=189788,819557,176485
BC00460=189788,819557,176485
BC00461=189788,819557,176485
BC00462=189788,819557,176483
BC00463=189788,819557,176483
BC00464=189788,819557,176483
BC00465=189788,819557,176483
BC00466=189788,819557,176486
BC00467=189788,819557,176486
BC00468=132304,777362,53
BC00469=132304,687429,53
BC00470=341619,775319,231168
BC00471=341619,843929,231168
BC00472=341619,843929,231168
BC00473=341015,843600,204386
BC00474=340773,843469,193674
BC00475=340773,843469,193674
BC00476=340773,843469,193674
BC00477=340773,843469,193674
BC00478=338609,842251,204386
BC00479=339214,842580,231168
BC00480=349631,842380,197374
BC00481=349631,842380,197374
BC00482=349631,842380,197374
BC00483=344838,853004,170892
BC00484=344838,853004,170892
BC00485=349631,842380,197374
BC00486=336550,839583,197374
BC00487=338313,841095,209130
BC00488=341619,843929,231168
BC00489=341619,775319,231168
BC00490=190901,728772,170929
BC00491=190901,786037,170929
BC00492=193011,793039,131574
BC00493=182032,791881,61669
BC00494=176016,791246,23364
BC00495=175802,792372,8727
BC00496=178212,792700,4465
BC00497=193011,793039,53
BC00498=193011,793039,53
BC00499=178212,792700,4465
BC00500=178845,792714,4276
BC00501=193612,789752,91438
BC00502=126346,753501,53
BC00503=70335,723316,53
BC00504=93918,779758,165352
BC00505=91695,784776,146437
BC00506=90805,786784,138870
BC00507=90805,786784,138870
BC00508=90805,786784,138870
BC00509=90805,786784,138870
BC00510=90805,786784,138870
BC00511=106862,787018,165353
BC00512=178185,787018,116808
BC00513=178185,787018,39086
BC00514=178185,787018,39086
BC00515=178185,787018,39086
BC00516=178185,787018,39086
BC00517=90805,786784,138870
BC00518=90805,786784,138870
BC00519=178185,787018,39086
BC00520=178185,787018,39086
BC00521=178185,787018,39085
BC00522=178185,787018,39085
BC00523=178185,787018,39085
BC00524=178185,787018,39085
BC00525=178185,787018,39085
EC00000=798156,0
EC00001=798156,0
EC00002=798156,0
EC00003=798156,0
EC00004=798156,0
EC00005=798156,0
EC00006=798156,0
EC00007=798155,1
EC00008=798155,1
EC00009=798155,1
EC00010=798155,1
EC00011=798155,1
EC00012=798155,1
EC00013=798155,1
EC00014=798155,1
EC00015=798155,1
EC00016=798155,1
EC00017=798155,1
EC00018=798155,1
EC00019=798155,1
EC00020=798155,1
EC00021=798155,1
EC00022=798154,1
EC00023=798154,1
EC00024=798154,1
EC00025=798154,1
EC00026=798154,1
EC00027=798153,2
EC00028=798153,2
EC00029=798153,2
EC00030=798153,2
EC00031=798153,2
EC00032=798153,2
EC00033=798153,2
EC00034=798153,2
EC00035=798153,2
EC00036=798153,2
EC00037=798153,2
EC00038=798153,2
EC00039=798153,2
EC00040=798153,2
EC00041=798153,2
EC00042=798154,2
EC00043=798155,1
EC00044=798156,0
EC00045=798156,0
EC00046=798156,0
EC00047=798156,0
EC00048=798156,0
EC00049=798153,0
EC00050=798153,0
EC00051=798153,0
EC00052=798153,0
EC00053=798153,0
EC00054=798153,0
EC00055=798153,0
EC00056=798153,0
EC00057=798153,0
EC00058=798153,0
EC00059=798153,0
EC00060=798153,0
EC00061=798153,0
EC00062=798153,0
EC00063=798153,0
EC00064=798153,0
EC00065=798153,0
EC00066=798152,0
EC00067=798152,0
EC00068=798152,0
EC00069=798152,0
EC00070=798152,0
EC00071=798152,0
EC00072=798152,0
EC00073=798152,0
EC00074=798152,0
EC00075=798152,0
EC00076=798152,0
EC00077=798152,0
EC00078=798152,0
EC00079=798152,0
EC00080=798152,0
EC00081=798152,0
EC00082=798152,0
EC00083=798150,0
EC00084=798150,0
EC00085=798150,0
EC00086=798150,0
EC00087=798150,0
EC00088=798150,0
EC00089=798150,0
EC00090=798150,0
EC00091=798150,0
EC00092=798149,1
EC00093=798149,1
EC00094=798149,1
EC00095=798149,1
EC00096=798149,1
EC00097=798149,1
EC00098=798149,1
EC00099=798149,1
EC00100=798149,1
EC00101=798156,0
EC00102=798156,0
EC00103=798156,0
EC00104=798156,0
EC00105=798156,0
EC00106=798156,0
EC00107=798156,0
EC00108=798156,0
EC00109=798156,0
EC00110=798156,0
EC00111=798156,0
EC00112=798156,0
EC00113=798156,0
EC00114=798156,0
EC00115=798156,0
EC00116=798156,0
EC00117=798156,0
EC00118=798156,0
EC00119=798156,0
EC00120=798155,0
EC00121=798155,0
EC00122=798155,0
EC00123=798155,0
EC00124=798155,0
EC00125=798155,0
EC00126=798155,0
EC00127=798155,0
EC00128=798155,0
EC00129=798155,0
EC00130=798155,0
EC00131=798155,0
EC00132=798155,0
EC00133=798155,0
EC00134=798156,0
EC00135=798156,0
EC00136=798156,0
EC00137=798156,0
EC00138=798156,0
EC00139=798156,0
EC00140=798156,0
EC00141=798156,0
EC00142=798156,0
EC00143=798156,0
EC00144=798156,0
EC00145=798156,0
EC00146=798156,0
EC00147=798156,0
EC00148=798156,0
EC00149=798156,0
EC00150=798156,0
EC00151=798156,0
EC00152=798156,0
EC00153=798156,0
EC00154=798156,0
EC00155=798156,0
EC00156=798156,0
EC00157=798156,0
EC00158=798156,0
EC00159=798156,0
EC00160=798156,0
EC00161=798156,0
EC00162=798156,0
EC00163=798156,0
EC00164=798156,0
EC00165=798156,0
EC00166=798156,0
EC00167=798156,0
EC00168=798156,0
EC00169=798156,0
EC00170=798156,0
EC00171=798156,0
EC00172=798156,0
EC00173=798156,0
EC00174=798156,0
EC00175=798156,0
EC00176=798156,0
EC00177=798156,0
EC00178=798156,0
EC00179=798156,0
EC00180=798156,0
EC00181=798156,0
EC00182=798156,0
EC00183=798156,0
EC00184=798156,0
EC00185=798156,0
EC00186=798156,0
EC00187=798156,0
EC00188=798156,0
EC00189=798156,0
EC00190=798156,0
EC00191=798156,0
EC00192=798156,0
EC00193=798156,0
EC00194=798156,0
EC00195=798156,0
EC00196=798156,0
EC00197=798156,0
EC00198=798156,0
EC00199=798156,0
EC00200=798156,0
EC00201=798156,0
EC00202=798156,0
EC00203=798156,0
EC00204=798156,0
EC00205=798156,0
EC00206=798156,0
EC00207=798156,0
EC00208=798156,0
EC00209=798156,0
EC00210=798156,0
EC00211=798156,0
EC00212=798156,0
EC00213=798156,0
EC00214=798156,0
EC00215=798156,0
EC00216=798156,0
EC00217=798156,0
EC00218=798156,0
EC00219=798156,0
EC00220=798156,0
EC00221=798156,0
EC00222=798156,0
EC00223=798156,0
EC00224=798156,0
EC00225=798156,0
EC00226=798156,0
EC00227=798156,0
EC00228=798156,0
EC00229=798156,0
EC00230=798156,0
EC00231=798156,0
EC00232=798156,0
EC00233=798156,0
EC00234=798156,0
EC00235=798156,0
EC00236=798156,0
EC00237=798156,0
EC00238=798156,0
EC00239=798154,0
EC00240=798154,0
EC00241=798154,0
EC00242=798154,0
EC00243=798154,0
EC00244=798154,0
EC00245=798154,0
EC00246=798154,0
EC00247=798154,0
EC00248=798154,0
EC00249=798154,0
EC00250=798154,0
EC00251=798154,0
EC00252=799965,0
EC00253=799965,0
EC00254=799965,0
EC00255=799965,0
EC00256=799965,0
EC00257=799965,0
EC00258=799962,1
EC00259=799962,1
EC00260=799962,1
EC00261=799960,2
EC00262=799960,2
EC00263=975524,0
EC00264=975524,0
EC00265=799958,2
EC00266=799958,2
EC00267=799958,2
EC00268=799958,2
EC00269=799958,2
EC00270=799958,2
EC00271=799958,2
EC00272=799958,2
EC00273=975524,0
EC00274=975524,0
EC00275=799958,2
EC00276=799958,2
EC00277=799958,2
EC00278=799958,2
EC00279=799958,2
EC00280=799958,2
EC00281=799955,2
EC00282=799955,2
EC00283=975524,0
EC00284=975524,0
EC00285=799955,2
EC00286=799955,2
EC00287=799955,2
EC00288=799955,2
EC00289=799954,3
EC00290=799951,3
EC00291=799951,3
EC00292=799951,3
EC00293=975524,0
EC00294=975524,0
EC00295=799951,3
EC00296=799951,3
EC00297=799951,3
EC00298=799951,3
EC00299=799951,3
EC00300=799951,3
EC00301=799951,3
EC00302=799951,3
EC00303=975524,0
EC00304=975524,0
EC00305=799951,3
EC00306=799949,4
EC00307=799950,4
EC00308=799951,3
EC00309=799951,3
EC00310=799951,3
EC00311=799951,3
EC00312=799951,3
EC00313=975524,0
EC00314=975524,0
EC00315=799951,3
EC00316=799951,3
EC00317=799951,3
EC00318=799951,3
EC00319=799951,3
EC00320=799951,3
EC00321=799951,3
EC00322=799951,3
EC00323=799951,3
EC00324=799951,3
EC00325=799949,3
EC00326=975524,0
EC00327=975524,0
EC00328=799949,3
EC00329=799949,3
EC00330=799949,3
EC00331=799949,3
EC00332=799949,3
EC00333=799949,3
EC00334=799949,3
EC00335=975524,0
EC00336=975524,0
EC00337=799949,3
EC00338=799949,3
EC00339=799949,3
EC00340=799949,3
EC00341=799949,3
EC00342=799949,3
EC00343=799949,3
EC00344=975524,0
EC00345=975524,0
EC00346=799949,3
EC00347=799949,3
EC00348=799949,3
EC00349=799949,3
EC00350=799949,3
EC00351=799949,3
EC00352=802129,3
EC00353=798156,0
EC00354=798156,0
EC00355=798156,0
EC00356=798156,0
EC00357=798156,0
EC00358=798156,0
EC00359=798156,0
EC00360=798156,0
EC00361=798156,0
EC00362=798156,0
EC00363=798156,0
EC00364=798156,0
EC00365=798156,0
EC00366=798156,0
EC00367=798156,0
EC00368=798156,0
EC00369=798156,0
EC00370=798156,0
EC00371=798156,0
EC00372=798156,0
EC00373=798156,0
EC00374=798156,0
EC00375=798156,0
EC00376=798156,0
EC00377=798156,0
EC00378=798156,0
EC00379=798156,0
EC00380=798156,0
EC00381=798156,0
EC00382=798156,0
EC00383=798156,0
EC00384=798156,0
EC00385=798156,0
EC00386=798156,0
EC00387=798156,0
EC00388=798156,0
EC00389=798156,0
EC00390=798156,0
EC00391=798153,2
EC00392=798153,2
EC00393=798153,2
EC00394=798153,2
EC00395=798153,2
EC00396=798153,2
EC00397=798153,2
EC00398=798153,2
EC00399=798153,2
EC00400=798153,2
EC00401=798153,2
EC00402=798153,2
EC00403=798152,2
EC00404=798153,2
EC00405=798153,2
EC00406=798153,2
EC00407=798153,2
EC00408=798153,2
EC00409=798156,0
EC00410=798156,0
EC00411=798156,0
EC00412=798156,0
EC00413=798156,0
EC00414=798156,0
EC00415=798156,0
EC00416=798156,0
EC00417=798156,0
EC00418=798156,0
EC00419=798156,0
EC00420=798156,0
EC00421=798156,0
EC00422=798156,0
EC00423=798156,0
EC00424=798156,0
EC00425=798156,0
EC00426=798156,0
EC00427=798156,0
EC00428=798156,0
EC00429=798156,0
EC00430=798156,0
EC00431=798156,0
EC00432=798156,0
EC00433=798156,0
EC00434=798156,0
EC00435=798156,0
EC00436=798156,0
EC00437=798156,0
EC00438=798156,0
EC00439=798156,0
EC00440=798156,0
EC00441=798156,0
EC00442=798156,0
EC00443=798156,0
EC00444=798152,0
EC00445=798152,0
EC00446=798152,0
EC00447=798152,0
EC00448=798152,0
EC00449=798152,0
EC00450=798152,0
EC00451=798152,0
EC00452=798152,0
EC00453=798152,0
EC00454=798152,0
EC00455=798152,0
EC00456=798152,0
EC00457=798152,0
EC00458=798152,0
EC00459=798152,0
EC00460=798152,0
EC00461=798152,0
EC00462=798152,0
EC00463=798152,0
EC00464=798152,0
EC00465=798152,0
EC00466=798152,0
EC00467=798152,0
EC00468=798156,0
EC00469=798156,0
EC00470=798156,0
EC00471=798156,0
EC00472=798156,0
EC00473=798156,0
EC00474=798156,0
EC00475=798156,0
EC00476=798156,0
EC00477=798156,0
EC00478=798156,0
EC00479=798156,0
EC00480=798156,0
EC00481=798156,0
EC00482=798155,1
EC00483=798156,0
EC00484=798156,0
EC00485=798156,0
EC00486=798156,0
EC00487=798156,0
EC00488=798156,0
EC00489=798156,0
EC00490=798156,0
EC00491=798156,0
EC00492=798156,0
EC00493=798156,0
EC00494=798156,0
EC00495=798156,0
EC00496=798156,0
EC00497=798156,0
EC00498=798156,0
EC00499=798156,0
EC00500=798156,0
EC00501=798156,0
EC00502=798156,0
EC00503=798156,0
EC00504=798156,0
EC00505=798156,0
EC00506=798156,0
EC00507=798156,0
EC00508=798156,0
EC00509=798156,0
EC00510=798156,0
EC00511=798156,0
EC00512=798156,0
EC00513=798156,0
EC00514=798156,0
EC00515=798156,0
EC00516=798156,0
EC00517=798156,0
EC00518=798156,0
EC00519=798156,0
EC00520=798156,0
EC00521=798155,0
EC00522=798155,0
EC00523=798155,0
EC00524=798155,0
EC00525=798155,0
///POSTYPE BASE
///RECTAN
///RCONF 0,0,0,0,0,0,0,0,0,0,0,0,0,0,0,0,0,0,0,0,0,0,0,0
P00006=0.222,-3.123,-1.508,0.0000,0.0000,0.0000
P00021=-0.225,-6.128,-0.405,0.0000,0.0000,0.0000
P00022=0.222,-3.123,-1.508,0.0000,0.0000,0.0000
P00023=0.143,-0.036,0.682,0.0000,0.0000,0.0000
P00024=0.145,-0.552,1.326,0.0000,0.0000,0.0000
P00025=-2.003,0.006,0.728,0.0000,0.0000,0.0000
P00026=0.562,-0.002,-0.337,0.0000,0.0000,0.0000
P00027=-0.746,0.015,-9.096,0.0000,0.0000,0.0000
P00028=-2.237,-0.018,-7.702,0.0000,0.0000,0.0000
P00029=-2.156,-0.086,-4.681,0.0000,0.0000,0.0000
P00030=5.926,-4.294,-1.390,0.0000,0.0000,0.0000
P00031=1.853,-0.001,-1.549,0.0000,0.0000,0.0000
P00032=1.957,0.503,-7.217,0.0000,0.0000,0.0000
///RCONF 0,0,0,0,1,0,0,0,0,0,0,0,0,0,0,0,0,0,0,0,0,0,0,0
P00033=-0.123,0.612,-5.012,0.0000,0.0000,0.0000
///RCONF 0,0,0,0,0,0,0,0,0,0,0,0,0,0,0,0,0,0,0,0,0,0,0,0
P00034=-0.304,0.773,-2.693,0.0000,0.0000,0.0000
P00035=2.817,0.591,-1.622,0.0000,0.0000,0.0000
P00036=-1.108,-0.829,1.850,0.0000,0.0000,0.0000
P00037=0.023,0.937,-2.677,0.0000,0.0000,0.0000
P00038=0.158,-1.133,-1.952,0.0000,0.0000,0.0000
P00039=0.012,-3.081,-0.106,0.0000,0.0000,0.0000
P00040=-0.030,9.648,2.467,0.0000,0.0000,0.0000
P00041=0.192,3.924,0.305,0.0000,0.0000,0.0000
P00042=-0.217,1.941,0.413,0.0000,0.0000,0.0000
P00043=-0.044,-1.937,1.197,0.0000,0.0000,0.0000
P00044=0.687,-2.322,1.156,0.0000,0.0000,0.0000
P00050=4.296,-4.501,-0.826,0.0000,0.0000,0.0000
P00051=0.367,3.892,0.009,0.0000,0.0000,0.0000
//INST
///DATE 2025/05/13 14:56
///ATTR SC,RW
///GROUP1 RB1,BS1
///GROUP2 ST1
NOP
'OK_r2_O38-47,64(2)(90,0)
'Down
MOVJ C00000 BC00000 VJ=100.00  +MOVJ EC00000 VJ=100.00
MOVJ C00001 BC00001 VJ=30.00  +MOVJ EC00001 VJ=100.00
'Path S1701
SFTOF3D
MOVJ C00002 BC00002 VJ=50.00  +MOVJ EC00002 VJ=100.00
MOVL C00003 BC00003 V=400.0  +MOVJ EC00003 VJ=100.00
SMOVL C00004 BC00004 V=166.7  +MOVJ EC00004
SREFP 3 C00005 BC00005  +REFP EC00005
CALL JOB:SEARCH-R1-S13D
SET P021 P006
SFTON3D P021
SMOVL C00006 BC00006 V=166.7  +MOVJ EC00006
SMOVL C00007 BC00007 V=166.7  +MOVJ EC00007
SMOVL C00008 BC00008 V=166.7  +MOVJ EC00008
SREFP 3 C00009 BC00009  +REFP EC00009
CALL JOB:SEARCH-R1-S13D
SET P021 P006
SFTON3D P021
SMOVL C00010 BC00010 V=166.7  +MOVJ EC00010
SREFP 3 C00011 BC00011  +REFP EC00011
CALL JOB:SEARCH-R1-S13D
SET P021 P006
SFTON3D P021
SMOVL C00012 BC00012 V=166.7  +MOVJ EC00012
SMOVL C00013 BC00013 V=166.7  +MOVJ EC00013
SMOVL C00014 BC00014 V=166.7  +MOVJ EC00014
SREFP 3 C00015 BC00015  +REFP EC00015
CALL JOB:SEARCH-R1-S13D
SET P021 P006
SFTON3D P021
SMOVL C00016 BC00016 V=166.7  +MOVJ EC00016
SFTOF3D
MOVJ C00017 BC00017 VJ=100.00  +MOVJ EC00017 VJ=100.00
MOVL C00018 BC00018 V=166.7  +MOVJ EC00018 VJ=100.00
MOVL C00019 BC00019 V=166.7  +MOVJ EC00019 VJ=100.00
MOVJ C00020 BC00020 VJ=100.00  +MOVJ EC00020 VJ=100.00
MOVL C00021 BC00021 V=166.7  +MOVJ EC00021 VJ=100.00
SMOVL C00022 BC00022 V=166.7  +MOVJ EC00022
SREFP 3 C00023 BC00023  +REFP EC00023
CALL JOB:SEARCH-R1-S13D
SET P024 P006
SFTON3D P024
SMOVL C00024 BC00024 V=166.7  +MOVJ EC00024
SREFP 3 C00025 BC00025  +REFP EC00025
CALL JOB:SEARCH-R1-S13D
SET P024 P006
SFTON3D P024
SMOVL C00026 BC00026 V=166.7  +MOVJ EC00026
SMOVL C00027 BC00027 V=166.7  +MOVJ EC00027
SREFP 3 C00028 BC00028  +REFP EC00028
CALL JOB:SEARCH-R1-S13D
SET P024 P006
SFTON3D P024
SMOVL C00029 BC00029 V=166.7  +MOVJ EC00029
MOVJ C00030 BC00030 VJ=50.00  +MOVJ EC00030 VJ=100.00
MOVL C00031 BC00031 V=166.7  +MOVJ EC00031 VJ=100.00
SMOVL C00032 BC00032 V=166.7  +MOVJ EC00032
SREFP 3 C00033 BC00033  +REFP EC00033
CALL JOB:SEARCH-R1-S13D
SET P025 P006
SFTON3D P025
SMOVL C00034 BC00034 V=166.7  +MOVJ EC00034
SREFP 3 C00035 BC00035  +REFP EC00035
CALL JOB:SEARCH-R1-S13D
SET P025 P006
SFTON3D P025
SMOVL C00036 BC00036 V=166.7  +MOVJ EC00036
SMOVL C00037 BC00037 V=166.7  +MOVJ EC00037
SREFP 3 C00038 BC00038  +REFP EC00038
CALL JOB:SEARCH-R1-S13D
SET P025 P006
SFTON3D P025
SMOVL C00039 BC00039 V=166.7  +MOVJ EC00039
SFTOF3D
SMOVL C00040 BC00040 V=166.7  +MOVJ EC00040
SMOVL C00041 BC00041 V=166.7  +MOVJ EC00041
SMOVL C00042 BC00042 V=166.7  +MOVJ EC00042
SMOVL C00043 BC00043 V=166.7  +MOVJ EC00043
MOVL C00044 BC00044 V=400.0  +MOVJ EC00044 VJ=100.00
MOVL C00045 BC00045 V=1000.0  +MOVJ EC00045 VJ=100.00
MOVJ C00046 BC00046 VJ=100.00  +MOVJ EC00046 VJ=100.00
MOVJ C00047 BC00047 VJ=100.00  +MOVJ EC00047 VJ=50.00
MOVL C00048 BC00048 V=1000.0  +MOVJ EC00048 VJ=100.00
MOVL C00049 BC00049 V=400.0  +MOVJ EC00049 VJ=100.00
SMOVL C00050 BC00050 V=166.7  +MOVJ EC00050
SREFP 3 C00051 BC00051  +REFP EC00051
CALL JOB:SEARCH-R1-S13D
SET P026 P006
SFTON3D P026
SMOVL C00052 BC00052 V=166.7  +MOVJ EC00052
SMOVL C00053 BC00053 V=166.7  +MOVJ EC00053
SMOVL C00054 BC00054 V=166.7  +MOVJ EC00054
SREFP 3 C00055 BC00055  +REFP EC00055
CALL JOB:SEARCH-R1-S13D
SET P026 P006
SFTON3D P026
SMOVL C00056 BC00056 V=166.7  +MOVJ EC00056
SFTOF3D
MOVL C00057 BC00057 V=400.0  +MOVJ EC00057 VJ=100.00
SMOVL C00058 BC00058 V=166.7  +MOVJ EC00058
SREFP 3 C00059 BC00059  +REFP EC00059
CALL JOB:SEARCH-R1-S13D
SET P027 P006
SFTON3D P027
SMOVL C00060 BC00060 V=166.7  +MOVJ EC00060
SMOVL C00061 BC00061 V=166.7  +MOVJ EC00061
SMOVL C00062 BC00062 V=166.7  +MOVJ EC00062
SREFP 3 C00063 BC00063  +REFP EC00063
CALL JOB:SEARCH-R1-S13D
SET P027 P006
SFTON3D P027
SMOVL C00064 BC00064 V=166.7  +MOVJ EC00064
SFTOF3D
MOVL C00065 BC00065 V=666.7  +MOVJ EC00065 VJ=100.00
SMOVL C00066 BC00066 V=166.7  +MOVJ EC00066
SREFP 3 C00067 BC00067  +REFP EC00067
CALL JOB:SEARCH-R1-S13D
SET P028 P006
SFTON3D P028
SMOVL C00068 BC00068 V=166.7  +MOVJ EC00068
SREFP 3 C00069 BC00069  +REFP EC00069
CALL JOB:SEARCH-R1-S13D
SET P028 P006
SFTON3D P028
SMOVL C00070 BC00070 V=166.7  +MOVJ EC00070
SMOVL C00071 BC00071 V=166.7  +MOVJ EC00071
SREFP 3 C00072 BC00072  +REFP EC00072
CALL JOB:SEARCH-R1-S13D
SET P028 P006
SFTON3D P028
SMOVL C00073 BC00073 V=166.7  +MOVJ EC00073
SFTOF3D
MOVL C00074 BC00074 V=333.3  +MOVJ EC00074 VJ=100.00
SMOVL C00075 BC00075 V=166.7  +MOVJ EC00075
SREFP 3 C00076 BC00076  +REFP EC00076
CALL JOB:SEARCH-R1-S13D
SET P029 P006
SFTON3D P029
SMOVL C00077 BC00077 V=166.7  +MOVJ EC00077
SREFP 3 C00078 BC00078  +REFP EC00078
CALL JOB:SEARCH-R1-S13D
SET P029 P006
SFTON3D P029
SMOVL C00079 BC00079 V=166.7  +MOVJ EC00079
SMOVL C00080 BC00080 V=166.7  +MOVJ EC00080
SREFP 3 C00081 BC00081  +REFP EC00081
CALL JOB:SEARCH-R1-S13D
SET P029 P006
SFTON3D P029
SMOVL C00082 BC00082 V=166.7  +MOVJ EC00082
SFTOF3D
MOVL C00083 BC00083 V=666.7  +MOVJ EC00083 VJ=100.00
SMOVL C00084 BC00084 V=166.7  +MOVJ EC00084
SREFP 3 C00085 BC00085  +REFP EC00085
CALL JOB:SEARCH-R1-S13D
SET P050 P006
SFTON3D P050
SMOVL C00086 BC00086 V=166.7  +MOVJ EC00086
SREFP 3 C00087 BC00087  +REFP EC00087
CALL JOB:SEARCH-R1-S13D
SET P050 P006
SFTON3D P050
SMOVL C00088 BC00088 V=166.7  +MOVJ EC00088
SMOVL C00089 BC00089 V=166.7  +MOVJ EC00089
SREFP 3 C00090 BC00090  +REFP EC00090
CALL JOB:SEARCH-R1-S13D
SET P050 P006
SFTON3D P050
SMOVL C00091 BC00091 V=166.7  +MOVJ EC00091
SFTOF3D
MOVL C00092 BC00092 V=333.3  +MOVJ EC00092 VJ=100.00
SMOVL C00093 BC00093 V=166.7  +MOVJ EC00093
SREFP 3 C00094 BC00094  +REFP EC00094
CALL JOB:SEARCH-R1-S13D
SET P051 P006
SFTON3D P051
SMOVL C00095 BC00095 V=166.7  +MOVJ EC00095
SREFP 3 C00096 BC00096  +REFP EC00096
CALL JOB:SEARCH-R1-S13D
SET P051 P006
SFTON3D P051
SMOVL C00097 BC00097 V=166.7  +MOVJ EC00097
SMOVL C00098 BC00098 V=166.7  +MOVJ EC00098
SREFP 3 C00099 BC00099  +REFP EC00099
CALL JOB:SEARCH-R1-S13D
SET P051 P006
SFTON3D P051
SMOVL C00100 BC00100 V=166.7  +MOVJ EC00100
SFTOF3D
MOVJ C00101 BC00101 VJ=100.00  +MOVJ EC00101 VJ=100.00
MOVJ C00102 BC00102 VJ=100.00  +MOVJ EC00102 VJ=100.00
MOVJ C00103 BC00103 VJ=100.00  +MOVJ EC00103 VJ=100.00
'Path S1702
SFTOF3D
MOVJ C00104 BC00104 VJ=100.00  +MOVJ EC00104 VJ=100.00
MOVL C00105 BC00105 V=166.7  +MOVJ EC00105 VJ=100.00
SMOVL C00106 BC00106 V=166.7  +MOVJ EC00106
SREFP 3 C00107 BC00107  +REFP EC00107
CALL JOB:SEARCH-R1-S13D
SET P022 P006
SFTON3D P022
SMOVL C00108 BC00108 V=166.7  +MOVJ EC00108
SMOVL C00109 BC00109 V=166.7  +MOVJ EC00109
SMOVL C00110 BC00110 V=166.7  +MOVJ EC00110
SREFP 3 C00111 BC00111  +REFP EC00111
CALL JOB:SEARCH-R1-S13D
SET P022 P006
SFTON3D P022
SMOVL C00112 BC00112 V=166.7  +MOVJ EC00112
SREFP 3 C00113 BC00113  +REFP EC00113
CALL JOB:SEARCH-R1-S13D
SET P022 P006
SFTON3D P022
SMOVL C00114 BC00114 V=166.7  +MOVJ EC00114
SMOVL C00115 BC00115 V=166.7  +MOVJ EC00115
SMOVL C00116 BC00116 V=166.7  +MOVJ EC00116
SREFP 3 C00117 BC00117  +REFP EC00117
CALL JOB:SEARCH-R1-S13D
SET P022 P006
SFTON3D P022
SMOVL C00118 BC00118 V=166.7  +MOVJ EC00118
SFTOF3D
MOVL C00119 BC00119 V=666.7  +MOVJ EC00119 VJ=100.00
SMOVL C00120 BC00120 V=666.7  +MOVJ EC00120
SMOVL C00121 BC00121 V=166.7  +MOVJ EC00121
SREFP 3 C00122 BC00122  +REFP EC00122
CALL JOB:SEARCH-R1-S13D
SET P032 P006
SFTON3D P032
SMOVL C00123 BC00123 V=166.7  +MOVJ EC00123
SMOVL C00124 BC00124 V=166.7  +MOVJ EC00124
SMOVL C00125 BC00125 V=166.7  +MOVJ EC00125
SREFP 3 C00126 BC00126  +REFP EC00126
CALL JOB:SEARCH-R1-S13D
SET P032 P006
SFTON3D P032
SMOVL C00127 BC00127 V=166.7  +MOVJ EC00127
SREFP 3 C00128 BC00128  +REFP EC00128
CALL JOB:SEARCH-R1-S13D
SET P032 P006
SFTON3D P032
SMOVL C00129 BC00129 V=166.7  +MOVJ EC00129
SMOVL C00130 BC00130 V=166.7  +MOVJ EC00130
SMOVL C00131 BC00131 V=166.7  +MOVJ EC00131
SREFP 3 C00132 BC00132  +REFP EC00132
CALL JOB:SEARCH-R1-S13D
SET P032 P006
SFTON3D P032
SMOVL C00133 BC00133 V=166.7  +MOVJ EC00133
SFTOF3D
SMOVL C00134 BC00134 V=500.0  +MOVJ EC00134
MOVL C00135 BC00135 V=1000.0  +MOVJ EC00135 VJ=100.00
MOVJ C00136 BC00136 VJ=100.00  +MOVJ EC00136 VJ=100.00
'Path S1703
SFTOF3D
MOVJ C00137 BC00137 VJ=100.00  +MOVJ EC00137 VJ=100.00
SMOVL C00138 BC00138 V=250.0  +MOVJ EC00138
SMOVL C00139 BC00139 V=100.0  +MOVJ EC00139
SREFP 3 C00140 BC00140  +REFP EC00140
CALL JOB:SEARCH-R1-S13D
SET P023 P006
SFTON3D P023
SMOVL C00141 BC00141 V=100.0  +MOVJ EC00141
SMOVL C00142 BC00142 V=100.0  +MOVJ EC00142
SREFP 3 C00143 BC00143  +REFP EC00143
CALL JOB:SEARCH-R1-S13D
SET P023 P006
SFTON3D P023
SMOVL C00144 BC00144 V=166.7  +MOVJ EC00144
MOVL C00145 BC00145 V=1000.0  +MOVJ EC00145 VJ=100.00
MOVL C00146 BC00146 V=1000.0  +MOVJ EC00146 VJ=100.00
MOVJ C00147 BC00147 VJ=100.00  +MOVJ EC00147 VJ=100.00
MOVJ C00148 BC00148 VJ=100.00  +MOVJ EC00148 VJ=100.00
MOVJ C00149 BC00149 VJ=100.00  +MOVJ EC00149 VJ=100.00
MOVJ C00150 BC00150 VJ=100.00  +MOVJ EC00150 VJ=100.00
MOVJ C00151 BC00151 VJ=100.00  +MOVJ EC00151 VJ=100.00
'Up
'Path S1246
SFTOF3D
MOVJ C00152 BC00152 VJ=100.00  +MOVJ EC00152 VJ=100.00
SMOVL C00153 BC00153 V=100.0  +MOVJ EC00153
SREFP 3 C00154 BC00154  +REFP EC00154
CALL JOB:SEARCH-R1-S13D
SET P030 P006
SFTON3D P030
SMOVL C00155 BC00155 V=100.0  +MOVJ EC00155
SREFP 3 C00156 BC00156  +REFP EC00156
CALL JOB:SEARCH-R1-S13D
SET P030 P006
SFTON3D P030
SMOVL C00157 BC00157 V=133.3  +MOVJ EC00157
SFTOF3D
MOVL C00158 BC00158 V=400.0  +MOVJ EC00158 VJ=100.00
SMOVL C00159 BC00159 V=100.0  +MOVJ EC00159
SREFP 3 C00160 BC00160  +REFP EC00160
CALL JOB:SEARCH-R1-S13D
SET P031 P006
SFTON3D P031
SMOVL C00161 BC00161 V=100.0  +MOVJ EC00161
SREFP 3 C00162 BC00162  +REFP EC00162
CALL JOB:SEARCH-R1-S13D
SET P031 P006
SFTON3D P031
SMOVL C00163 BC00163 V=133.3  +MOVJ EC00163
MOVL C00164 BC00164 V=1000.0  +MOVJ EC00164 VJ=100.00
'Path S1276
SFTOF3D
COMM PAUSE
COMM MOVJ C00165 BC00165 VJ=100.00  +MOVJ EC00165 VJ=100.00
COMM MOVL C00166 BC00166 V=400.0  +MOVJ EC00166 VJ=100.00
COMM SMOVL C00167 BC00167 V=100.0  +MOVJ EC00167
COMM SREFP 3 C00168 BC00168  +REFP EC00168
COMM CALL JOB:SEARCH-R1-S13D
COMM SET P032 P006
COMM SFTON3D P032
COMM SMOVL C00169 BC00169 V=100.0  +MOVJ EC00169
COMM SREFP 3 C00170 BC00170  +REFP EC00170
COMM CALL JOB:SEARCH-R1-S13D
COMM SET P032 P006
COMM SFTON3D P032
COMM SMOVL C00171 BC00171 V=100.0  +MOVJ EC00171
COMM MOVL C00172 BC00172 V=400.0  +MOVJ EC00172 VJ=100.00
COMM SFTOF3D
COMM MOVJ C00173 BC00173 VJ=100.00  +MOVJ EC00173 VJ=100.00
COMM SMOVL C00174 BC00174 V=100.0  +MOVJ EC00174
COMM SREFP 3 C00175 BC00175  +REFP EC00175
COMM CALL JOB:SEARCH-R1-S13D
COMM SET P033 P006
COMM SFTON3D P033
COMM SMOVL C00176 BC00176 V=100.0  +MOVJ EC00176
COMM SREFP 3 C00177 BC00177  +REFP EC00177
COMM CALL JOB:SEARCH-R1-S13D
COMM SET P033 P006
COMM SFTON3D P033
COMM SMOVL C00178 BC00178 V=100.0  +MOVJ EC00178
COMM SFTOF3D
COMM MOVL C00179 BC00179 V=400.0  +MOVJ EC00179 VJ=100.00
MOVJ C00180 BC00180 VJ=100.00  +MOVJ EC00180 VJ=100.00
SMOVL C00181 BC00181 V=100.0  +MOVJ EC00181
SREFP 3 C00182 BC00182  +REFP EC00182
CALL JOB:SEARCH-R1-S13D
SET P034 P006
SFTON3D P034
SMOVL C00183 BC00183 V=100.0  +MOVJ EC00183
SREFP 3 C00184 BC00184  +REFP EC00184
CALL JOB:SEARCH-R1-S13D
SET P034 P006
SFTON3D P034
SMOVL C00185 BC00185 V=100.0  +MOVJ EC00185
MOVL C00186 BC00186 V=400.0  +MOVJ EC00186 VJ=100.00
MOVJ C00187 BC00187 VJ=100.00  +MOVJ EC00187 VJ=100.00
'Path S1278
SFTOF3D
MOVJ C00188 BC00188 VJ=100.00  +MOVJ EC00188 VJ=100.00
SMOVL C00189 BC00189 V=100.0  +MOVJ EC00189
SREFP 3 C00190 BC00190  +REFP EC00190
CALL JOB:SEARCH-R1-S13D
SET P035 P006
SFTON3D P035
SMOVL C00191 BC00191 V=100.0  +MOVJ EC00191
SREFP 3 C00192 BC00192  +REFP EC00192
CALL JOB:SEARCH-R1-S13D
SET P035 P006
SFTON3D P035
SMOVL C00193 BC00193 V=100.0  +MOVJ EC00193
SFTOF3D
MOVL C00194 BC00194 V=400.0  +MOVJ EC00194 VJ=100.00
SMOVL C00195 BC00195 V=100.0  +MOVJ EC00195
SREFP 3 C00196 BC00196  +REFP EC00196
CALL JOB:SEARCH-R1-S13D
SET P036 P006
SFTON3D P036
SMOVL C00197 BC00197 V=100.0  +MOVJ EC00197
SREFP 3 C00198 BC00198  +REFP EC00198
CALL JOB:SEARCH-R1-S13D
SET P036 P006
SFTON3D P036
SMOVL C00199 BC00199 V=100.0  +MOVJ EC00199
'Path S1970
SFTOF3D
MOVJ C00200 BC00200 VJ=100.00  +MOVJ EC00200 VJ=100.00
MOVL C00201 BC00201 V=400.0  +MOVJ EC00201 VJ=100.00
SMOVL C00202 BC00202 V=100.0  +MOVJ EC00202
SREFP 3 C00203 BC00203  +REFP EC00203
CALL JOB:SEARCH-R1-S13D
SET P037 P006
SFTON3D P037
SMOVL C00204 BC00204 V=100.0  +MOVJ EC00204
SREFP 3 C00205 BC00205  +REFP EC00205
CALL JOB:SEARCH-R1-S13D
SET P037 P006
SFTON3D P037
SMOVL C00206 BC00206 V=100.0  +MOVJ EC00206
SFTOF3D
MOVL C00207 BC00207 V=400.0  +MOVJ EC00207 VJ=100.00
MOVL C00208 BC00208 V=1000.0  +MOVJ EC00208 VJ=100.00
COMM PAUSE
COMM MOVJ C00209 BC00209 VJ=100.00  +MOVJ EC00209 VJ=100.00
COMM SMOVL C00210 BC00210 V=100.0  +MOVJ EC00210
COMM SREFP 3 C00211 BC00211  +REFP EC00211
COMM CALL JOB:SEARCH-R1-S13D
COMM SET P038 P006
COMM SFTON3D P038
COMM SMOVL C00212 BC00212 V=100.0  +MOVJ EC00212
COMM SREFP 3 C00213 BC00213  +REFP EC00213
COMM CALL JOB:SEARCH-R1-S13D
COMM SET P038 P006
COMM SFTON3D P038
COMM SMOVL C00214 BC00214 V=100.0  +MOVJ EC00214
COMM SFTOF3D
COMM MOVL C00215 BC00215 V=400.0  +MOVJ EC00215 VJ=100.00
COMM SMOVL C00216 BC00216 V=100.0  +MOVJ EC00216
COMM SREFP 3 C00217 BC00217  +REFP EC00217
COMM CALL JOB:SEARCH-R1-S13D
COMM SET P039 P006
COMM SFTON3D P039
COMM SMOVL C00218 BC00218 V=100.0  +MOVJ EC00218
COMM SREFP 3 C00219 BC00219  +REFP EC00219
COMM CALL JOB:SEARCH-R1-S13D
COMM SET P039 P006
COMM SFTON3D P039
COMM SMOVL C00220 BC00220 V=100.0  +MOVJ EC00220
COMM MOVJ C00221 BC00221 VJ=100.00  +MOVJ EC00221 VJ=100.00
SFTOF3D
MOVJ C00222 BC00222 VJ=100.00  +MOVJ EC00222 VJ=100.00
MOVJ C00223 BC00223 VJ=100.00  +MOVJ EC00223 VJ=100.00
MOVJ C00224 BC00224 VJ=100.00  +MOVJ EC00224 VJ=100.00
MOVJ C00225 BC00225 VJ=100.00  +MOVJ EC00225 VJ=100.00
SMOVL C00226 BC00226 V=100.0  +MOVJ EC00226
SREFP 3 C00227 BC00227  +REFP EC00227
CALL JOB:SEARCH-R1-S13D
SET P040 P006
SFTON3D P040
SMOVL C00228 BC00228 V=100.0  +MOVJ EC00228
SREFP 3 C00229 BC00229  +REFP EC00229
CALL JOB:SEARCH-R1-S13D
SET P040 P006
SFTON3D P040
SMOVL C00230 BC00230 V=100.0  +MOVJ EC00230
SFTOF3D
MOVL C00231 BC00231 V=1000.0  +MOVJ EC00231 VJ=100.00
SMOVL C00232 BC00232 V=100.0  +MOVJ EC00232
SREFP 3 C00233 BC00233  +REFP EC00233
CALL JOB:SEARCH-R1-S13D
SET P041 P006
SFTON3D P041
SMOVL C00234 BC00234 V=100.0  +MOVJ EC00234
SREFP 3 C00235 BC00235  +REFP EC00235
CALL JOB:SEARCH-R1-S13D
SET P041 P006
SFTON3D P041
SMOVL C00236 BC00236 V=100.0  +MOVJ EC00236
MOVJ C00237 BC00237 VJ=100.00  +MOVJ EC00237 VJ=100.00
SFTOF3D
MOVJ C00238 BC00238 VJ=100.00  +MOVJ EC00238 VJ=100.00
MOVL C00239 BC00239 V=400.0  +MOVJ EC00239 VJ=100.00
SMOVL C00240 BC00240 V=100.0  +MOVJ EC00240
SREFP 3 C00241 BC00241  +REFP EC00241
CALL JOB:SEARCH-R1-S13D
SET P042 P006
SFTON3D P042
SMOVL C00242 BC00242 V=100.0  +MOVJ EC00242
SREFP 3 C00243 BC00243  +REFP EC00243
CALL JOB:SEARCH-R1-S13D
SET P042 P006
SFTON3D P042
SMOVL C00244 BC00244 V=100.0  +MOVJ EC00244
SFTOF3D
MOVL C00245 BC00245 V=400.0  +MOVJ EC00245 VJ=100.00
'Path S1282
SFTOF3D
SMOVL C00246 BC00246 V=100.0  +MOVJ EC00246
SREFP 3 C00247 BC00247  +REFP EC00247
CALL JOB:SEARCH-R1-S13D
SET P043 P006
SFTON3D P043
SMOVL C00248 BC00248 V=100.0  +MOVJ EC00248
SREFP 3 C00249 BC00249  +REFP EC00249
CALL JOB:SEARCH-R1-S13D
SET P043 P006
SFTON3D P043
SMOVL C00250 BC00250 V=100.0  +MOVJ EC00250
SFTOF3D
MOVL C00251 BC00251 V=400.0  +MOVJ EC00251 VJ=100.00
MOVL C00252 BC00252 V=1000.0  +MOVJ EC00252 VJ=100.00
MOVJ C00253 BC00253 VJ=100.00  +MOVJ EC00253 VJ=100.00
MOVJ C00254 BC00254 VJ=100.00  +MOVJ EC00254 VJ=100.00
MOVL C00255 BC00255 V=400.0  +MOVJ EC00255 VJ=100.00
SMOVL C00256 BC00256 V=100.0  +MOVJ EC00256
SREFP 3 C00257 BC00257  +REFP EC00257
CALL JOB:SEARCH-R1-S13D
SET P044 P006
SFTON3D P044
SMOVL C00258 BC00258 V=100.0  +MOVJ EC00258
SREFP 3 C00259 BC00259  +REFP EC00259
CALL JOB:SEARCH-R1-S13D
SET P044 P006
SFTON3D P044
SMOVL C00260 BC00260 V=100.0  +MOVJ EC00260
MOVL C00261 BC00261 V=400.0  +MOVJ EC00261 VJ=100.00
SFTON3D P044
SMOVL C00262 BC00262 V=133.3 PL=0  +MOVJ EC00262
SREFP 1 C00263 BC00263  +REFP EC00263
SREFP 2 C00264 BC00264  +REFP EC00264
MACRO1 MJ#(0) ARGF9
ARCON
SWVON WEV#(60)
SMOVL C00265 BC00265 V=8.3  +MOVJ EC00265
SMOVL C00266 BC00266 V=8.3  +MOVJ EC00266
SMOVL C00267 BC00267 V=8.3  +MOVJ EC00267
ARCOF
SWVOF
SMOVL C00268 BC00268 V=250.0  +MOVJ EC00268
SFTOF3D
MOVJ C00269 BC00269 VJ=100.00  +MOVJ EC00269 VJ=100.00
SFTOF3D
MOVJ C00270 BC00270 VJ=70.00  +MOVJ EC00270 VJ=100.00
'Path W1138
MOVJ C00271 BC00271 VJ=100.00  +MOVJ EC00271 VJ=100.00
SFTOF
SFTON3D P037
SMOVL C00272 BC00272 V=133.3 PL=0  +MOVJ EC00272
SREFP 1 C00273 BC00273  +REFP EC00273
SREFP 2 C00274 BC00274  +REFP EC00274
MACRO1 MJ#(0) ARGF9
ARCON
SWVON WEV#(60)
SMOVL C00275 BC00275 V=8.3  +MOVJ EC00275
SMOVL C00276 BC00276 V=8.3  +MOVJ EC00276
SMOVL C00277 BC00277 V=8.3  +MOVJ EC00277
ARCOF
SWVOF
SMOVL C00278 BC00278 V=400.0  +MOVJ EC00278
MOVJ C00279 BC00279 VJ=100.00  +MOVJ EC00279 VJ=100.00
SFTOF3D
COMM PAUSE
COMM MOVJ C00280 BC00280 VJ=100.00  +MOVJ EC00280 VJ=100.00
COMM MOVJ C00281 BC00281 VJ=100.00  +MOVJ EC00281 VJ=100.00
COMM SFTON3D P039
COMM SMOVL C00282 BC00282 V=133.3 PL=0  +MOVJ EC00282
COMM SREFP 1 C00283 BC00283  +REFP EC00283
COMM SREFP 2 C00284 BC00284  +REFP EC00284
COMM MACRO1 MJ#(0) ARGF14
COMM ARCON
COMM SFTON3D P038
COMM SMOVL C00285 BC00285 V=8.3  +MOVJ EC00285
COMM SMOVL C00286 BC00286 V=8.3  +MOVJ EC00286
COMM ARCOF
COMM SMOVL C00287 BC00287 V=400.0  +MOVJ EC00287
COMM SFTOF3D
COMM MOVJ C00288 BC00288 VJ=100.00  +MOVJ EC00288 VJ=100.00
COMM MOVJ C00289 BC00289 VJ=100.00  +MOVJ EC00289 VJ=100.00
COMM MOVJ C00290 BC00290 VJ=100.00  +MOVJ EC00290 VJ=100.00
COMM MOVJ C00291 BC00291 VJ=100.00  +MOVJ EC00291 VJ=100.00
COMM 'Path W1140
COMM SFTOF3D
COMM SFTON3D P033
COMM SMOVL C00292 BC00292 V=133.3 PL=0  +MOVJ EC00292
COMM SREFP 1 C00293 BC00293  +REFP EC00293
COMM SREFP 2 C00294 BC00294  +REFP EC00294
COMM MACRO1 MJ#(0) ARGF14
COMM ARCON
COMM SWVON WEV#(10)
COMM SMOVL C00295 BC00295 V=8.3  +MOVJ EC00295
COMM SFTON3D P032
COMM SMOVL C00296 BC00296 V=8.3  +MOVJ EC00296
COMM SMOVL C00297 BC00297 V=8.3  +MOVJ EC00297
COMM ARCOF
COMM SWVOF
COMM SMOVL C00298 BC00298 V=400.0  +MOVJ EC00298
COMM SFTOF3D
COMM MOVJ C00299 BC00299 VJ=100.00  +MOVJ EC00299 VJ=100.00
SFTOF3D
MOVJ C00300 BC00300 VJ=100.00  +MOVJ EC00300 VJ=100.00
'Path W1142
SFTOF3D
SFTON3D P030
MOVJ C00301 BC00301 VJ=100.00  +MOVJ EC00301 VJ=100.00
SMOVL C00302 BC00302 V=133.3 PL=0  +MOVJ EC00302
SREFP 1 C00303 BC00303  +REFP EC00303
SREFP 2 C00304 BC00304  +REFP EC00304
MACRO1 MJ#(0) ARGF9
ARCON
SMOVL C00305 BC00305 V=8.3  +MOVJ EC00305
SFTON3D P031
SMOVL C00306 BC00306 V=8.3  +MOVJ EC00306
SMOVL C00307 BC00307 V=8.3  +MOVJ EC00307
SMOVL C00308 BC00308 V=8.3  +MOVJ EC00308
ARCOF
SMOVL C00309 BC00309 V=400.0  +MOVJ EC00309
SFTOF3D
MOVJ C00310 BC00310 VJ=100.00  +MOVJ EC00310 VJ=100.00
'Path W1143
SFTOF3D
SFTON3D P034
MOVJ C00311 BC00311 VJ=100.00  +MOVJ EC00311 VJ=100.00
SMOVL C00312 BC00312 V=133.3 PL=0  +MOVJ EC00312
SREFP 1 C00313 BC00313  +REFP EC00313
SREFP 2 C00314 BC00314  +REFP EC00314
MACRO1 MJ#(0) ARGF9
ARCON
SMOVC C00315 BC00315 V=8.3  +MOVJ EC00315
SMOVC C00316 BC00316 V=8.3  +MOVJ EC00316
SMOVC C00317 BC00317 V=8.3  +MOVJ EC00317
SMOVL C00318 BC00318 V=8.3  +MOVJ EC00318
SMOVC C00319 BC00319 V=8.3  +MOVJ EC00319
SMOVC C00320 BC00320 V=8.3  +MOVJ EC00320
SMOVC C00321 BC00321 V=8.3  +MOVJ EC00321
ARCOF
SMOVL C00322 BC00322 V=400.0  +MOVJ EC00322
SFTOF3D
MOVJ C00323 BC00323 VJ=100.00  +MOVJ EC00323 VJ=100.00
'Path W1144
SFTOF3D
SFTON3D P036
MOVJ C00324 BC00324 VJ=100.00  +MOVJ EC00324 VJ=100.00
SFTON3D P036
SMOVL C00325 BC00325 V=133.3 PL=0  +MOVJ EC00325
SREFP 1 C00326 BC00326  +REFP EC00326
SREFP 2 C00327 BC00327  +REFP EC00327
MACRO1 MJ#(0) ARGF14
ARCON
SMOVL C00328 BC00328 V=9.2  +MOVJ EC00328
SFTON3D P035
SMOVL C00329 BC00329 V=9.2  +MOVJ EC00329
SMOVL C00330 BC00330 V=9.2  +MOVJ EC00330
ARCOF
SMOVL C00331 BC00331 V=400.0  +MOVJ EC00331
SFTOF3D
MOVJ C00332 BC00332 VJ=100.00  +MOVJ EC00332 VJ=100.00
MOVJ C00333 BC00333 VJ=100.00  +MOVJ EC00333 VJ=100.00
SFTON3D P042
SMOVL C00334 BC00334 V=133.3 PL=0  +MOVJ EC00334
SREFP 1 C00335 BC00335  +REFP EC00335
SREFP 2 C00336 BC00336  +REFP EC00336
MACRO1 MJ#(0) ARGF14
ARCON
SMOVL C00337 BC00337 V=10.0  +MOVJ EC00337
SFTON3D P043
SMOVL C00338 BC00338 V=10.0  +MOVJ EC00338
SMOVL C00339 BC00339 V=10.0  +MOVJ EC00339
ARCOF
SMOVL C00340 BC00340 V=400.0  +MOVJ EC00340
MOVJ C00341 BC00341 VJ=100.00  +MOVJ EC00341 VJ=100.00
MOVJ C00342 BC00342 VJ=100.00  +MOVJ EC00342 VJ=100.00
SFTOF3D
SFTON3D P040
SMOVL C00343 BC00343 V=133.3 PL=0  +MOVJ EC00343
SREFP 1 C00344 BC00344  +REFP EC00344
SREFP 2 C00345 BC00345  +REFP EC00345
MACRO1 MJ#(0) ARGF14
ARCON
SMOVL C00346 BC00346 V=10.0  +MOVJ EC00346
SFTON3D P041
SMOVL C00347 BC00347 V=10.0  +MOVJ EC00347
SMOVL C00348 BC00348 V=10.0  +MOVJ EC00348
ARCOF
SMOVL C00349 BC00349 V=400.0  +MOVJ EC00349
SFTOF3D
MOVJ C00350 BC00350 VJ=100.00  +MOVJ EC00350 VJ=100.00
MOVJ C00351 BC00351 VJ=100.00  +MOVJ EC00351 VJ=100.00
MOVJ C00352 BC00352 VJ=100.00  +MOVJ EC00352 VJ=100.00
MOVJ C00353 BC00353 VJ=100.00  +MOVJ EC00353 VJ=100.00
MOVJ C00354 BC00354 VJ=100.00  +MOVJ EC00354 VJ=100.00
'Down
'1
MOVJ C00355 BC00355 VJ=100.00  +MOVJ EC00355 VJ=100.00
'Path W1705
SFTOF3D
SFTON3D P023
MOVJ C00356 BC00356 VJ=100.00  +MOVJ EC00356 VJ=100.00
SMOVL C00357 BC00357 V=400.0  +MOVJ EC00357
SMOVL C00358 BC00358 V=133.3 PL=0  +MOVJ EC00358
SREFP 1 C00359 BC00359  +REFP EC00359
SREFP 2 C00360 BC00360  +REFP EC00360
MACRO1 MJ#(0) ARGF14
ARCON
SMOVL C00361 BC00361 V=10.0  +MOVJ EC00361
SMOVL C00362 BC00362 V=10.0  +MOVJ EC00362
SMOVL C00363 BC00363 V=10.0  +MOVJ EC00363
ARCOF
SMOVL C00364 BC00364 V=400.0  +MOVJ EC00364
SMOVL C00365 BC00365 V=1000.0  +MOVJ EC00365
SFTOF3D
MOVJ C00366 BC00366 VJ=100.00  +MOVJ EC00366 VJ=100.00
MOVJ C00367 BC00367 VJ=100.00  +MOVJ EC00367 VJ=100.00
'2
MOVJ C00368 BC00368 VJ=100.00  +MOVJ EC00368 VJ=100.00
MOVJ C00369 BC00369 VJ=100.00  +MOVJ EC00369 VJ=100.00
MOVJ C00370 BC00370 VJ=100.00  +MOVJ EC00370 VJ=100.00
'Path W1706
SFTOF3D
SFTON3D P021
MOVJ C00371 BC00371 VJ=15.00  +MOVJ EC00371 VJ=100.00
SMOVL C00372 BC00372 V=400.0  +MOVJ EC00372
SMOVL C00373 BC00373 V=100.0 PL=0  +MOVJ EC00373
SREFP 1 C00374 BC00374  +REFP EC00374
SREFP 2 C00375 BC00375  +REFP EC00375
MACRO1 MJ#(0) ARGF14
ARCON
SMOVL C00376 BC00376 V=10.0  +MOVJ EC00376
ARCOF
SMOVL C00377 BC00377 V=400.0  +MOVJ EC00377
SMOVL C00378 BC00378 V=1000.0  +MOVJ EC00378
SFTOF3D
MOVJ C00379 BC00379 VJ=50.00  +MOVJ EC00379 VJ=100.00
'Path W1707
SFTOF3D
SFTON3D P021
MOVJ C00380 BC00380 VJ=100.00  +MOVJ EC00380 VJ=100.00
SMOVL C00381 BC00381 V=400.0  +MOVJ EC00381
SMOVL C00382 BC00382 V=100.0 PL=0  +MOVJ EC00382
SREFP 1 C00383 BC00383  +REFP EC00383
SREFP 2 C00384 BC00384  +REFP EC00384
MACRO1 MJ#(0) ARGF14
ARCON
SMOVL C00385 BC00385 V=10.0  +MOVJ EC00385
ARCOF
SMOVL C00386 BC00386 V=400.0  +MOVJ EC00386
SMOVL C00387 BC00387 V=1000.0  +MOVJ EC00387
SFTOF3D
SMOVL C00388 BC00388 V=500.0  +MOVJ EC00388
SMOVL C00389 BC00389 V=500.0  +MOVJ EC00389
SMOVL C00390 BC00390 V=400.0  +MOVJ EC00390
SMOVL C00391 BC00391 V=166.7  +MOVJ EC00391
MOVJ C00392 BC00392 VJ=50.00  +MOVJ EC00392 VJ=100.00
MOVL C00393 BC00393 V=166.7  +MOVJ EC00393 VJ=100.00
MOVL C00394 BC00394 V=166.7  +MOVJ EC00394 VJ=0.78
SFTON3D P024
MACRO1 MJ#(0) ARGF9
SMOVL C00395 BC00395 V=150.0 PL=0  +MOVJ EC00395
ARCON
SFTON3D P025
SMOVL C00396 BC00396 V=11.7  +MOVJ EC00396
SMOVC C00397 BC00397 V=13.3  +MOVJ EC00397
SMOVC C00398 BC00398 V=13.3  +MOVJ EC00398
SMOVC C00399 BC00399 V=13.3  +MOVJ EC00399
SFTON3D P024
SMOVL C00400 BC00400 V=11.7  +MOVJ EC00400
SMOVL C00401 BC00401 V=11.7  +MOVJ EC00401
SMOVC C00402 BC00402 V=13.3  +MOVJ EC00402
SMOVC C00403 BC00403 V=13.3  +MOVJ EC00403
SMOVC C00404 BC00404 V=13.3  +MOVJ EC00404
ARCOF
SMOVL C00405 BC00405 V=333.3  +MOVJ EC00405
SFTOF3D
MOVL C00406 BC00406 V=333.3  +MOVJ EC00406 VJ=0.78
MOVL C00407 BC00407 V=333.3  +MOVJ EC00407 VJ=0.78
MOVL C00408 BC00408 V=333.3  +MOVJ EC00408 VJ=0.78
MOVJ C00409 BC00409 VJ=100.00  +MOVJ EC00409 VJ=100.00
MOVJ C00410 BC00410 VJ=100.00  +MOVJ EC00410 VJ=100.00
'3
MOVJ C00411 BC00411 VJ=100.00  +MOVJ EC00411 VJ=100.00
MOVJ C00412 BC00412 VJ=100.00  +MOVJ EC00412 VJ=100.00
'Path W1709
SFTOF3D
SFTON3D P023
MOVJ C00413 BC00413 VJ=100.00  +MOVJ EC00413 VJ=100.00
SMOVL C00414 BC00414 V=400.0  +MOVJ EC00414
SMOVL C00415 BC00415 V=133.3 PL=0  +MOVJ EC00415
SREFP 1 C00416 BC00416  +REFP EC00416
SREFP 2 C00417 BC00417  +REFP EC00417
MACRO1 MJ#(0) ARGF14
ARCON
SMOVL C00418 BC00418 V=10.0  +MOVJ EC00418
SMOVL C00419 BC00419 V=10.0  +MOVJ EC00419
SMOVL C00420 BC00420 V=10.0  +MOVJ EC00420
ARCOF
SMOVL C00421 BC00421 V=400.0  +MOVJ EC00421
SMOVL C00422 BC00422 V=1000.0  +MOVJ EC00422
SFTOF3D
MOVJ C00423 BC00423 VJ=100.00  +MOVJ EC00423 VJ=100.00
MOVJ C00424 BC00424 VJ=100.00  +MOVJ EC00424 VJ=100.00
'4
MOVJ C00425 BC00425 VJ=100.00  +MOVJ EC00425 VJ=100.00
MOVJ C00426 BC00426 VJ=100.00  +MOVJ EC00426 VJ=100.00
'Path W1710
SFTOF3D
SFTON3D P032
MOVJ C00427 BC00427 VJ=15.00  +MOVJ EC00427 VJ=100.00
SMOVL C00428 BC00428 V=400.0  +MOVJ EC00428
SMOVL C00429 BC00429 V=133.3 PL=0  +MOVJ EC00429
SREFP 1 C00430 BC00430  +REFP EC00430
SREFP 2 C00431 BC00431  +REFP EC00431
MACRO1 MJ#(0) ARGF14
ARCON
SMOVL C00432 BC00432 V=10.0  +MOVJ EC00432
ARCOF
SMOVL C00433 BC00433 V=400.0  +MOVJ EC00433
SMOVL C00434 BC00434 V=1000.0  +MOVJ EC00434
SFTOF3D
'Path W1711
SFTOF3D
SFTON3D P032
MOVJ C00435 BC00435 VJ=100.00  +MOVJ EC00435 VJ=100.00
SMOVL C00436 BC00436 V=400.0  +MOVJ EC00436
SMOVL C00437 BC00437 V=133.3 PL=0  +MOVJ EC00437
SREFP 1 C00438 BC00438  +REFP EC00438
SREFP 2 C00439 BC00439  +REFP EC00439
MACRO1 MJ#(0) ARGF14
ARCON
SMOVL C00440 BC00440 V=10.0  +MOVJ EC00440
ARCOF
SMOVL C00441 BC00441 V=400.0  +MOVJ EC00441
SMOVL C00442 BC00442 V=1000.0  +MOVJ EC00442
SFTOF3D
MOVJ C00443 BC00443 VJ=100.00  +MOVJ EC00443 VJ=100.00
MOVL C00444 BC00444 V=666.7  +MOVJ EC00444 VJ=100.00
SFTON3D P028
MACRO1 MJ#(0) ARGF9
SMOVL C00445 BC00445 V=150.0 PL=0  +MOVJ EC00445
ARCON
SFTON3D P029
SMOVL C00446 BC00446 V=11.7  +MOVJ EC00446
SMOVC C00447 BC00447 V=13.3  +MOVJ EC00447
SMOVC C00448 BC00448 V=13.3  +MOVJ EC00448
SMOVC C00449 BC00449 V=13.3  +MOVJ EC00449
SFTON3D P028
SMOVL C00450 BC00450 V=11.7  +MOVJ EC00450
SMOVL C00451 BC00451 V=11.7  +MOVJ EC00451
SMOVC C00452 BC00452 V=13.3  +MOVJ EC00452
SMOVC C00453 BC00453 V=13.3  +MOVJ EC00453
SMOVC C00454 BC00454 V=13.3  +MOVJ EC00454
ARCOF
SMOVL C00455 BC00455 V=333.3  +MOVJ EC00455
SFTOF3D
MOVL C00456 BC00456 V=666.7  +MOVJ EC00456 VJ=100.00
SFTON3D P051
MACRO1 MJ#(0) ARGF9
SMOVL C00457 BC00457 V=150.0 PL=0  +MOVJ EC00457
ARCON
SFTON3D P050
SMOVL C00458 BC00458 V=11.7  +MOVJ EC00458
SMOVC C00459 BC00459 V=13.3  +MOVJ EC00459
SMOVC C00460 BC00460 V=13.3  +MOVJ EC00460
SMOVC C00461 BC00461 V=13.3  +MOVJ EC00461
SFTON3D P051
SMOVL C00462 BC00462 V=11.7  +MOVJ EC00462
SMOVL C00463 BC00463 V=11.7  +MOVJ EC00463
SMOVC C00464 BC00464 V=13.3  +MOVJ EC00464
SMOVC C00465 BC00465 V=13.3  +MOVJ EC00465
SMOVC C00466 BC00466 V=13.3  +MOVJ EC00466
ARCOF
SMOVL C00467 BC00467 V=333.3  +MOVJ EC00467
SFTOF3D
MOVJ C00468 BC00468 VJ=100.00  +MOVJ EC00468 VJ=100.00
MOVJ C00469 BC00469 VJ=100.00  +MOVJ EC00469 VJ=100.00
'6
MOVJ C00470 BC00470 VJ=100.00  +MOVJ EC00470 VJ=100.00
MOVJ C00471 BC00471 VJ=100.00  +MOVJ EC00471 VJ=100.00
'Path W1714
SFTOF3D
SFTON3D P022
MOVJ C00472 BC00472 VJ=100.00  +MOVJ EC00472 VJ=100.00
SMOVL C00473 BC00473 V=400.0  +MOVJ EC00473
SMOVL C00474 BC00474 V=133.3 PL=0  +MOVJ EC00474
SREFP 1 C00475 BC00475  +REFP EC00475
SREFP 2 C00476 BC00476  +REFP EC00476
MACRO1 MJ#(0) ARGF14
ARCON
SMOVL C00477 BC00477 V=10.0  +MOVJ EC00477
ARCOF
SMOVL C00478 BC00478 V=400.0  +MOVJ EC00478
SMOVL C00479 BC00479 V=1000.0  +MOVJ EC00479
SFTOF3D
'Path W1715
SFTOF3D
SFTON3D P022
MOVJ C00480 BC00480 VJ=100.00  +MOVJ EC00480 VJ=100.00
SMOVL C00481 BC00481 V=400.0  +MOVJ EC00481
SMOVL C00482 BC00482 V=133.3 PL=0  +MOVJ EC00482
SREFP 1 C00483 BC00483  +REFP EC00483
SREFP 2 C00484 BC00484  +REFP EC00484
MACRO1 MJ#(0) ARGF14
ARCON
SFTON3D P032
SMOVL C00485 BC00485 V=10.0  +MOVJ EC00485
ARCOF
SMOVL C00486 BC00486 V=400.0  +MOVJ EC00486
SFTOF3D
MOVJ C00487 BC00487 VJ=100.00  +MOVJ EC00487 VJ=14.00
MOVJ C00488 BC00488 VJ=100.00  +MOVJ EC00488 VJ=100.00
MOVJ C00489 BC00489 VJ=100.00  +MOVJ EC00489 VJ=100.00
MOVJ C00490 BC00490 VJ=100.00  +MOVJ EC00490 VJ=100.00
MOVJ C00491 BC00491 VJ=100.00  +MOVJ EC00491 VJ=100.00
'7
MOVJ C00492 BC00492 VJ=100.00  +MOVJ EC00492 VJ=100.00
'Path W1716
SFTOF3D
SFTON3D P022
MOVJ C00493 BC00493 VJ=100.00  +MOVJ EC00493 VJ=25.00
MOVJ C00494 BC00494 VJ=100.00  +MOVJ EC00494 VJ=100.00
SMOVL C00495 BC00495 V=400.0  +MOVJ EC00495
SMOVL C00496 BC00496 V=133.3 PL=0  +MOVJ EC00496
SREFP 1 C00497 BC00497  +REFP EC00497
SREFP 2 C00498 BC00498  +REFP EC00498
MACRO1 MJ#(0) ARGF14
ARCON
SMOVL C00499 BC00499 V=11.7  +MOVJ EC00499
ARCOF
SMOVL C00500 BC00500 V=400.0  +MOVJ EC00500
SFTOF3D
MOVJ C00501 BC00501 VJ=50.00  +MOVJ EC00501 VJ=100.00
MOVJ C00502 BC00502 VJ=100.00  +MOVJ EC00502 VJ=25.00
MOVJ C00503 BC00503 VJ=30.00  +MOVJ EC00503 VJ=100.00
'Path W1717
SFTOF3D
SFTON3D P022
MOVJ C00504 BC00504 VJ=30.00  +MOVJ EC00504 VJ=100.00
SMOVL C00505 BC00505 V=400.0  +MOVJ EC00505
SMOVL C00506 BC00506 V=133.3 PL=0  +MOVJ EC00506
SREFP 1 C00507 BC00507  +REFP EC00507
SREFP 2 C00508 BC00508  +REFP EC00508
MACRO1 MJ#(0) ARGF14
ARCON
SMOVL C00509 BC00509 V=11.7  +MOVJ EC00509
ARCOF
SMOVL C00510 BC00510 V=400.0  +MOVJ EC00510
SFTOF3D
SMOVL C00511 BC00511 V=1000.0  +MOVJ EC00511
SMOVL C00512 BC00512 V=1000.0  +MOVJ EC00512
SMOVL C00513 BC00513 V=1000.0  +MOVJ EC00513
SMOVL C00514 BC00514 V=1000.0  +MOVJ EC00514
SFTON3D P027
SMOVL C00515 BC00515 V=1000.0  +MOVJ EC00515
SMOVL C00516 BC00516 V=133.3 PL=0  +MOVJ EC00516
SREFP 1 C00517 BC00517  +REFP EC00517
SREFP 2 C00518 BC00518  +REFP EC00518
MACRO1 MJ#(0) ARGF9
ARCON
SMOVL C00519 BC00519 V=11.7  +MOVJ EC00519
SMOVL C00520 BC00520 V=11.7  +MOVJ EC00520
SFTON3D P026
SMOVL C00521 BC00521 V=11.7  +MOVJ EC00521
SMOVL C00522 BC00522 V=11.7  +MOVJ EC00522
ARCOF
SMOVL C00523 BC00523 V=400.0  +MOVJ EC00523
SFTOF3D
SMOVL C00524 BC00524 V=500.0  +MOVJ EC00524
SMOVL C00525 BC00525 V=500.0  +MOVJ EC00525
END
